# B&R Automation Studio project Y4_V3_1 (part 5)

#### ConBuffersCyclic.st - Cyclic code
```iecst
(********************************************************************
 * COPYRIGHT --
 ********************************************************************
 * Program: ConSeam2
 * File: ConSeam2Cyclic.st
 * Author: nicke
 ********************************************************************
 * Implementation of program ConSeam2
 ********************************************************************)

PROGRAM _CYCLIC

   //TRACKINGSECTION END BLOCK CONDITIONS
	Tracking30.Blocks[0] := (Tracking40.Busy) ;
	Tracking30.Blocks[2] := (CB2.Input.Fault) ;
	Tracking30.Blocks[9] := (S16Photo.Int) ;
	Tracking30.Blocks[10] := (S17Photo.Int) ;
	Tracking30.ControlIN := Control.Achieved1 ;
	Tracking30.EMOStart := EMO.StartLatch ;
	Tracking30.ESClear := Control.ESClear ;
	Tracking30 ();
	Tracking30.ResMan := FALSE ;
	Tracking30.BlockInhib := (Tracking41.Busy) AND NOT(Tracking40.Busy) ;
	CASE Tracking30.Index OF
		0: //RESET ALL TRACKBIT FOR SELECTED TRACKINGSECTION
			Track301 := TrackClear ;
			Track302 := TrackClear ;
		1: //TRACK FROM NOT Tracking20.Blocked (-) TO S14Photo.Int (P)
			Track302 := TrackClear ;
			//FB INPUTS
			Track301.FixedIN := Tracking30.FixedOUT ;
			Track301.Speed := Speeds.SpeedExit ;
			Track301.TimeoutEN := TRUE ;
			Track301.TimeoutACK := Warn.Ack ;
			Track301.TimeoutBlock := (Warn.Block) ;
			Track301.DelayPT := TrackDelayPT.PTTrack301 ;
			//FB CALL
			Track301 ();
			//FB OUTPUTS
			CB1.o.Run[0] := Track301.RunOUT ;
			CB1.Inv.Scale1.x := Track301.SpeedOUT ;
			IF(Track301.Done) THEN
				Tracking30.IndexIN := 2 ;
			END_IF
		2: //TRACK FROM S14Photo.Int (P) TO NOT Tracking30.Blocked (-)
			Track301 := TrackClear ;
			//FB INPUTS
			Track302.FixedIN := Tracking30.FixedOUT ;
			//FB CALL
			Track302 ();
			//FB OUTPUTS
			IF(Track302.Done) THEN
				Tracking30.IndexIN := 0 ;
				Tracking40.IndexIN := 1 ;
				Tracking93.IndexIN := 1 ;
				Tracking40.LengthIN := Tracking30.Length ;
				Tracking40.WidthIN := Tracking30.Width ;
				Tracking40.RowBlockIN := Tracking30.RowBlock ;
			END_IF
	END_CASE

	//TRACKBIT DONE CONDITIONS
	Track301.DoneIN := EDGEPOS(S14Photo.Int) ;
	Track302.DoneIN := NOT(Tracking30.Blocked) ;

	//TRACKINGSECTION END BLOCK CONDITIONS
	Tracking93.ControlIN := Control.Achieved1 ;
	Tracking93.EMOStart := EMO.StartLatch ;
	Tracking93.ESClear := Control.ESClear ;
	Tracking93 ();
	Tracking93.ResMan := FALSE ;
	CASE Tracking93.Index OF
		0: //RESET ALL TRACKBIT FOR SELECTED TRACKINGSECTION
			Track931 := TrackClear ;
			Track932 := TrackClear ;
		1: //TRACK FROM NOT Tracking30.Blocked (-) TO S15Photo.Int (N)
			Track932 := TrackClear ;
			//FB INPUTS
			Track931.FixedIN := Tracking93.FixedOUT ;
			Track931.RunBlock := (Track401.TimeoutOUT) OR(Track402.TimeoutOUT) ;
			Track931.Speed := Speeds.SpeedExit ;
			//FB CALL
			Track931 ();
			//FB OUTPUTS
			CB1.o.Run[0] := Track931.RunOUT ;
			CB1.Inv.Scale1.x := Track931.SpeedOUT ;
			IF(Track931.Done) THEN
				Tracking93.IndexIN := 2 ;
			END_IF
		2: //TRACK FROM S15Photo.Int (N) TO Track932.DelayTON.Q (P)
			Track931 := TrackClear ;
			//FB INPUTS
			Track932.FixedIN := Tracking93.FixedOUT ;
			Track932.RunBlock := (Track401.TimeoutOUT) OR(Track402.TimeoutOUT) ;
			Track932.Speed := Speeds.SpeedExit ;
			Track932.TrackDelayEN := TRUE ;
			Track932.DelayPT := TrackDelayPT.PTTrack932 ;
			//FB CALL
			Track932 ();
			//FB OUTPUTS
			CB1.o.Run[0] := Track932.RunOUT ;
			CB1.Inv.Scale1.x := Track932.SpeedOUT ;
			IF(Track932.Done) THEN
				Tracking93.IndexIN := 0 ;
			END_IF
	END_CASE

	//TRACKBIT DONE CONDITIONS
	Track931.DoneIN := EDGENEG(S15Photo.Int) ;

	//MANUAL RESET CONDITIONS FOR CONCURRENT TRACKBIT
	Tracking93.ResMan := Tracking40.ResMan ;
	IF(Tracking40.IndexIN = 0) THEN
		Tracking93.IndexIN := 0 ;
	END_IF
	IF EDGEPOS(Track302.Active)AND((Track401.Active)OR(Track402.Active))THEN
		Tracking93.IndexIN:=0;
	END_IF

	//TRACKINGSECTION END BLOCK CONDITIONS
	Tracking40.Blocks[0] := (Tracking41.Busy) OR(S58Lever.In ) OR(S58Lever.Int) OR(Tracking51.Busy) ;
	Tracking40.Blocks[1] := (Tracking50.IndexIN > 1) OR(Tracking52.Busy) ;
	Tracking40.Blocks[2] := (RowTemp.Done) ;
	Tracking40.Blocks[4] := NOT(Sol33Pal4.Auto) ;
	Tracking40.Blocks[9] := (S17Photo.Int) ;
	Tracking40.Blocks[10] := (S18Photo.Int) ;
	Tracking40.Blocks[11] := NOT(S37Reed.In) ;
	Tracking40.ControlIN := Control.Achieved1 ;
	Tracking40.EMOStart := EMO.StartLatch ;
	Tracking40.ESClear := Control.ESClear ;
	Tracking40 ();
	Tracking40.ResMan := FALSE ;
	CASE Tracking40.Index OF
		0: //RESET ALL TRACKBIT FOR SELECTED TRACKINGSECTION
			Track401 := TrackClear ;
			Track402 := TrackClear ;
		1: //TRACK FROM NOT Tracking30.Blocked (-) TO S16Photo.Int (P)
			Track402 := TrackClear ;
			//FB INPUTS
			Track401.FixedIN := Tracking40.FixedOUT ;
			Track401.Speed := Speeds.SpeedExit ;
			Track401.TimeoutEN := TRUE ;
			Track401.TimeoutACK := Warn.Ack ;
			Track401.TimeoutBlock := (Warn.Block) ;
			Track401.DelayPT := TrackDelayPT.PTTrack401 ;
			//FB CALL
			Track401 ();
			//FB OUTPUTS
			CB2.o.Run[0] := Track401.RunOUT ;
			CB2.Inv.Scale1.x := Track401.SpeedOUT ;
			IF(Track401.Done) THEN
				Tracking40.IndexIN := 2 ;
			END_IF
		2: //TRACK FROM S16Photo.Int (P) TO NOT Tracking40.Blocked (-)
			Track401 := TrackClear ;
			//FB INPUTS
			Track402.FixedIN := Tracking40.FixedOUT ;
			//FB CALL
			Track402 ();
			//FB OUTPUTS
			IF(Track402.Done) THEN
				Tracking40.IndexIN := 0 ;
				IF NOT(Tracking40.Blocked) THEN
					Tracking41.IndexIN := 1 ;
				ELSE
					Tracking41.IndexIN := 2 ;
				END_IF
				Tracking41.LengthIN := Tracking40.Length ;
				Tracking41.WidthIN := Tracking40.Width ;
				Tracking41.RowBlockIN := Tracking40.RowBlock ;
			END_IF
	END_CASE

	//TRACKBIT DONE CONDITIONS
	Track401.DoneIN := EDGEPOS(S16Photo.Int) ;
	Track402.DoneIN := NOT(Tracking40.Blocked) ;

	//TRACKINGSECTION END BLOCK CONDITIONS
	Tracking41.ControlIN := Control.Achieved1 ;
	Tracking41.EMOStart := EMO.StartLatch ;
	Tracking41.ESClear := Control.ESClear ;
	Tracking41 ();
	Tracking41.ResMan := FALSE ;
	CASE Tracking41.Index OF
		0: //RESET ALL TRACKBIT FOR SELECTED TRACKINGSECTION
			Track411 := TrackClear ;
			Track412 := TrackClear ;
			Track413 := TrackClear ;
			Track414 := TrackClear ;
		1: //TRACK FROM NOT Tracking40.Blocked (-) TO Track411.DelayTON.Q (P)
			Track412 := TrackClear ;
			Track413 := TrackClear ;
			Track414 := TrackClear ;
			//FB INPUTS
			Track411.FixedIN := Tracking41.FixedOUT ;
			Track411.Speed := Speeds.SpeedExit ;
			Track411.TrackDelayEN := TRUE ;
			Track411.DelayPT := TrackDelayPT.PTTrack411 ;
			//FB CALL
			Track411 ();
			//FB OUTPUTS
			CB2.o.Run[0] := Track411.RunOUT ;
			CB2.Inv.Scale1.x := Track411.SpeedOUT ;
			IF(Track411.Done) THEN
				Tracking41.IndexIN := 2 ;
			END_IF
		2: //TRACK FROM Track411.DelayTON.Q (P) TO S17Photo.Int (N)
			Track411 := TrackClear ;
			Track413 := TrackClear ;
			Track414 := TrackClear ;
			//FB INPUTS
			Track412.FixedIN := Tracking41.FixedOUT ;
			Track412.Speed := Speeds.SpeedExit ;
			Track412.TimeoutEN := TRUE ;
			Track412.TimeoutACK := Warn.Ack ;
			Track412.TimeoutBlock := (Warn.Block) ;
			Track412.DelayPT := TrackDelayPT.PTTrack412 ;
			//FB CALL
			Track412 ();
			//FB OUTPUTS
			CB2.o.Run[0] := Track412.RunOUT ;
			CRB.o.Run[0] := Track412.RunOUT ;
			CB2.Inv.Scale1.x := Track412.SpeedOUT ;
			CRB.Inv.Scale1.x := Track412.SpeedOUT ;
			IF(Track412.Done) THEN
				Tracking41.IndexIN := 3 ;
			END_IF
		3: //TRACK FROM S17Photo.Int (N) TO S17Photo.Int (P)
			Track411 := TrackClear ;
			Track412 := TrackClear ;
			Track414 := TrackClear ;
			//FB INPUTS
			Track413.FixedIN := Tracking41.FixedOUT ;
			Track413.Speed := Speeds.SpeedSlow ;
			Track413.TimeoutEN := TRUE ;
			Track413.TimeoutACK := Warn.Ack ;
			Track413.TimeoutBlock := (Warn.Block) ;
			Track413.DelayPT := TrackDelayPT.PTTrack413 ;
			//FB CALL
			Track413 ();
			//FB OUTPUTS
			CRB.o.Rev[0] := Track413.RunOUT ;
			CRB.Inv.Scale1.x := Track413.SpeedOUT ;
			IF(Track413.Done) THEN
				Tracking41.IndexIN := 4 ;
			END_IF
		4: //TRACK FROM S17Photo.Int (P) TO S17Photo.Int (N)
			Track411 := TrackClear ;
			Track412 := TrackClear ;
			Track413 := TrackClear ;
			//FB INPUTS
			Track414.FixedIN := Tracking41.FixedOUT ;
			Track414.Speed := Speeds.SpeedSlow ;
			//FB CALL
			Track414 ();
			//FB OUTPUTS
			CRB.o.Run[0] := Track414.RunOUT ;
			CRB.Inv.Scale1.x := Track414.SpeedOUT ;
			IF(Track414.Done) THEN
				Tracking41.IndexIN := 0 ;
				Tracking50.IndexIN := 1 ;
				Tracking50.RowBlockIN := Tracking41.RowBlock ;
			END_IF
	END_CASE

	//TRACKBIT DONE CONDITIONS
	Track412.DoneIN := EDGENEG(S17Photo.Int) ;
	Track413.DoneIN := EDGEPOS(S17Photo.Int) ;
	Track414.DoneIN := EDGENEG(S17Photo.Int) ;

END_PROGRAM
```

### Program Logical/Automatic/ConRow (IEC) - Row Building Conveyor

#### ConRowCyclic.st - Cyclic code
```iecst
(********************************************************************
 * COPYRIGHT --
 ********************************************************************
 * Program: ConRowBuild
 * File: ConRowBuildCyclic.st
 * Author: nicke
 ********************************************************************
 * Implementation of program ConRowBuild
 ********************************************************************)

PROGRAM _CYCLIC

   //TRACKINGSECTION END BLOCK CONDITIONS
	Tracking50.Blocks[0] := (Tracking60.Index > 1) ;
	Tracking50.Blocks[1] := Tracking70.Busy ;
	Tracking50.Blocks[2] := (CRE.Input.Fault) ;
	Tracking50.Blocks[3] := (CLB.Input.Fault) ;
	Tracking50.Blocks[9] := (S19Photo.Int) ;
//	Tracking50.Blocks[10] := (S20Photo.Int) ;
	Tracking50.Blocks[11] := (S21Photo.Int) ;
	Tracking50.ControlIN := Control.Achieved1 ;
	Tracking50.EMOStart := EMO.StartLatch ;
	Tracking50.ESClear := Control.ESClear ;
	Tracking50 ();
	IF(Tracking50.ResMan) OR(Tracking50.ResES) THEN
		Rows.Tracking50 := Rows.Empty ;
	END_IF
	Tracking50.ResMan := FALSE ;
	//RESET OF OUTPUTS
	Sol33Pal4.Auto := TRUE ;
	CASE Tracking50.Index OF
		0: //RESET ALL TRACKBIT FOR SELECTED TRACKINGSECTION
			Track501 := TrackClear ;
			Track502 := TrackClear ;
			Track503 := TrackClear ;
			Track504 := TrackClear ;
			Track505 := TrackClear ;
			Track506 := TrackClear ;
			Track507 := TrackClear ;
		1: //TRACK FROM S17Photo.Int (N) TO RowTemp.Done (P)
			Track502 := TrackClear ;
			Track503 := TrackClear ;
			Track504 := TrackClear ;
			Track505 := TrackClear ;
			Track506 := TrackClear ;
			Track507 := TrackClear ;
			//FB INPUTS
			Track501.FixedIN := Tracking50.FixedOUT ;
			//FB CALL
			Track501 ();
			//FB OUTPUTS
			IF(Track501.Done) THEN
				Tracking50.IndexIN := 2 ;
			END_IF
		2: //TRACK FROM RowTemp.Done (P) TO Track502.DelayTON.Q (P)
			Track501 := TrackClear ;
			Track503 := TrackClear ;
			Track504 := TrackClear ;
			Track505 := TrackClear ;
			Track506 := TrackClear ;
			Track507 := TrackClear ;
			//FB INPUTS
			Track502.FixedIN := Tracking50.FixedOUT ;
			Track502.Speed := Speeds.SpeedCntr ;
			Track502.TrackDelayEN := TRUE ;
			Track502.DelayPT := TrackDelayPT.PTTrack502 ;
			//FB CALL
			Track502 ();
			//FB OUTPUTS
			CRB.o.Run[0] := Track502.RunOUT ;
			CRB.Inv.Scale1.x := Track502.SpeedOUT ;
			IF(S18Photo.Int) THEN
				Track502.DoneIN := TRUE ;
			END_IF
			IF(Track502.Done) THEN
				IF NOT(Tracking50.RowBlock)THEN // Furnace 1
					Tracking50.IndexIN := 3 ;
				ELSE // Furnace 2
					Tracking50.IndexIN := 0 ;
					Tracking52.IndexIN := 3 ;
					Tracking52.LengthIN := Tracking50.Length ;
					Tracking52.BatchClearIN := Tracking50.BatchClear;
				END_IF
			END_IF
		3: //TRACK FROM Track502.DelayTON.Q (P) TO S36Reed.In (P)
			Track501 := TrackClear ;
			Track502 := TrackClear ;
			Track504 := TrackClear ;
			Track505 := TrackClear ;
			Track506 := TrackClear ;
			Track507 := TrackClear ;
			//FB INPUTS
			Track503.FixedIN := Tracking50.FixedOUT ;
			Track503.SolBlock := (Tracking50.Blocked) ;
			Track503.TimeoutEN := TRUE ;
			Track503.TimeoutACK := Warn.Ack ;
			Track503.TimeoutBlock := (Warn.Block) ;
			Track503.DelayPT := TrackDelayPT.PTTrack503 ;
			//FB CALL
			Track503 ();
			//FB OUTPUTS
			Sol33Pal4.Auto := NOT(Track503.SolOUT) ;
			IF(Track503.Done) THEN
				Tracking50.IndexIN := 4 ;
			END_IF
		4: //TRACK FROM S36Reed.In (P) TO S19Photo.Int (P)
			Track501 := TrackClear ;
			Track502 := TrackClear ;
			Track503 := TrackClear ;
			Track505 := TrackClear ;
			Track506 := TrackClear ;
			Track507 := TrackClear ;
			//FB INPUTS
			Track504.FixedIN := Tracking50.FixedOUT ;
			Track504.Speed := Speeds.SpeedBatch ;
			Track504.TimeoutEN := TRUE ;
			Track504.TimeoutACK := Warn.Ack ;
			Track504.TimeoutBlock := (Warn.Block) ;
			Track504.DelayPT := TrackDelayPT.PTTrack504 ;
			//FB CALL
			Track504 ();
			//FB OUTPUTS
			CRE.o.Run[0] := Track504.RunOUT ;
			CRE.Inv.Scale1.x := Track504.SpeedOUT ;
			Sol33Pal4.Auto := NOT(Track504.SolOUT) ;
			IF(Track504.Done) THEN
				Tracking50.IndexIN := 5 ;
			END_IF
		5: //TRACK FROM S19Photo.Int (P) TO Track505.DelayTON.Q (N)
			Track501 := TrackClear ;
			Track502 := TrackClear ;
			Track503 := TrackClear ;
			Track504 := TrackClear ;
			Track506 := TrackClear ;
			Track507 := TrackClear ;
			//FB INPUTS
			Track505.FixedIN := Tracking50.FixedOUT ;
			Track505.Speed := Speeds.SpeedBatch ;
			Track505.TrackDelayEN := TRUE ;
			Track505.DelayPT := TrackDelayPT.PTTrack505 ;
			//FB CALL
			Track505 ();
			//FB OUTPUTS
			CRE.o.Run[0] := Track505.RunOUT ;
			CRE.Inv.Scale1.x := Track505.SpeedOUT ;
			Sol33Pal4.Auto := NOT(Track505.SolOUT) ;
			IF(Track505.Done) THEN
				Tracking50.IndexIN := 6 ;
			END_IF
		6: //TRACK FROM Track505.DelayTON.Q (P) TO S19Photo.Int (N)
			Track501 := TrackClear ;
			Track502 := TrackClear ;
			Track503 := TrackClear ;
			Track504 := TrackClear ;
			Track505 := TrackClear ;
			Track507 := TrackClear ;
			//FB INPUTS
			Track506.FixedIN := Tracking50.FixedOUT ;
			Track506.Speed := Speeds.SpeedBatch ;
			Track506.TimeoutEN := TRUE ;
			Track506.TimeoutACK := Warn.Ack ;
			Track506.TimeoutBlock := (Warn.Block) ;
			Track506.DelayPT := TrackDelayPT.PTTrack506 ;
			//FB CALL
			Track506 ();
			//FB OUTPUTS
			CRE.o.Run[0] := Track506.RunOUT ;
			CLB.o.Run[0] := Track506.RunOUT ;
			CRE.Inv.Scale1.x := Track506.SpeedOUT ;
			CLB.Inv.Scale1.x := Track506.SpeedOUT ;
			Sol33Pal4.Auto := NOT(Track506.SolOUT) ;
			IF(Track506.Done) THEN
				Tracking50.IndexIN := 7 ;
			END_IF
		7: //TRACK FROM S19Photo.Int (N) TO Track507.DelayTON.Q (P)
			Track501 := TrackClear ;
			Track502 := TrackClear ;
			Track503 := TrackClear ;
			Track504 := TrackClear ;
			Track505 := TrackClear ;
			Track506 := TrackClear ;
			//FB INPUTS
			Track507.FixedIN := Tracking50.FixedOUT ;
			Track507.Speed := Speeds.SpeedSlow ;
			Track507.TrackDelayEN := TRUE ;
			Track507.DelayPT := TrackDelayPT.PTTrack507 ;
			//FB CALL
			Track507 ();
			//FB OUTPUTS
			CRE.o.Run[0] := Track507.RunOUT ;
			CLB.o.Run[0] := Track507.RunOUT ;
			CRE.Inv.Scale1.x := Track507.SpeedOUT ;
			CLB.Inv.Scale1.x := Track507.SpeedOUT ;
			IF(Track507.Done) THEN
				Tracking50.IndexIN := 0 ;
				Tracking60.IndexIN := 1 ;
				Tracking60.BatchClearIN := Tracking50.BatchClear ;
			END_IF
	END_CASE

	//TRACKBIT DONE CONDITIONS
	Track501.DoneIN := EDGEPOS(RowTemp.Done) ;
	Track503.DoneIN := EDGEPOS(S36Reed.In) ;
	Track504.DoneIN := EDGEPOS(S19Photo.Int) ;
	Track506.DoneIN := EDGENEG(S19Photo.Int) ;

	//TRACKINGSECTION END BLOCK CONDITIONS
	Tracking52.Blocks[0] := NOT(AGVReady.In) ;
	Tracking52.Blocks[1] := NOT(AGVInPosition.In) ;
	Tracking52.ControlIN := Control.Achieved1 ;
	Tracking52.EMOStart := EMO.StartLatch ;
	Tracking52.ESClear := Control.ESClear ;
	Tracking52 ();
	Tracking52.ResMan := FALSE ;
	//RESET OF OUTPUTS
	AGVReadyToSend.Auto := FALSE ;
	AGVSending.Auto := FALSE ;
	AGVBatchClear.Auto := FALSE;
	CASE Tracking52.Index OF
		0: //RESET ALL TRACKBIT FOR SELECTED TRACKINGSECTION
			Track521 := TrackClear ;
			Track522 := TrackClear ;
		1: //TRACK FROM Track502.DelayTON.Q (P) TO NOT(Tracking52.Blocked) (-)
			Track522 := TrackClear ;
			//FB INPUTS
			Track521.FixedIN := Tracking52.FixedOUT ;
			//FB CALL
			Track521 ();
			//FB OUTPUTS
			AGVReadyToSend.Auto := Track521.SolOUT ;
			IF(Track521.Done) THEN
				Tracking52.IndexIN := 2 ;
			END_IF
		2: //TRACK FROM NOT(Tracking52.Blocked) (-)  TO Track522.DelayTON.Q (P)
			Track521 := TrackClear ;
			//FB INPUTS
			Track522.FixedIN := Tracking52.FixedOUT ;
			//Track522.Speed := Speeds.SpeedBatch ; //SSS
			Track522.Speed := Speeds.SpeedTrans ; //SSS
			Track522.TrackDelayEN := TRUE ;
			Track522.DelayPT := TrackDelayPT.PTTrack805 ;
			//FB CALL
			Track522 ();
			//FB OUTPUTS
			AGVReadyToSend.Auto := Track522.SolOUT ;
			AGVSending.Auto := Track522.RunOUT ;
			AGVBatchClear.Auto := Tracking52.BatchClear;
			CRB.o.Run[0] := Track522.RunOUT ;
			CRB.Inv.Scale1.x := Track522.SpeedOUT ;
			IF(Track522.Done) THEN
				Tracking52.IndexIN := 0 ;
			END_IF
		3://Trick to beat the problem of Track521.DoneIN being true when IndexIN = 1.
			Tracking52.IndexIN := 1 ;
	END_CASE

	//TRACKBIT DONE CONDITIONS
	Track521.DoneIN := NOT(Tracking52.Blocked) ;

	AGVRequired.Auto := FALSE;
	IF(Tracking10.RowBlock) OR(Tracking11.RowBlock) OR(Tracking20.RowBlock) OR(Tracking30.RowBlock) OR(Tracking40.RowBlock) OR(Tracking50.RowBlock)THEN
		AGVRequired.Auto := TRUE;
	END_IF
END_PROGRAM
```

### Program Logical/Automatic/ConBatch (IEC) - Batch Building Conveyor

#### ConBatchCyclic.st - Cyclic code
```iecst
(********************************************************************
 * COPYRIGHT --
 ********************************************************************
 * Program: ConBatch
 * File: ConBatchCyclic.st
 * Author: nicke
 ********************************************************************
 * Implementation of program ConBatch
 ********************************************************************)

PROGRAM _CYCLIC

  //TRACKINGSECTION END BLOCK CONDITIONS
	Tracking60.Blocks[9] := (Pause.Active) ;
	Tracking60.Blocks[10] := NOT(WashRun.In) ;
	Tracking60.Blocks[11] := NOT(FurnReady.Int) ;
	Tracking60.Blocks[12] := (S55Lever.In) ;
	Tracking60.ControlIN := Control.Achieved1 ;
	Tracking60.EMOStart := EMO.StartLatch ;
	Tracking60.ESClear := Control.ESClear ;
	Tracking60 ();
	IF(Tracking60.ResMan) OR(Tracking60.ResES) THEN
		Loads.AshtonExit := Loads.Empty ;
	END_IF
	Tracking60.ResMan := FALSE ;
	//RESET OF OUTPUTS
	BatchAtExit.Auto := FALSE ;
	WashStop.Auto := FALSE ;
	CASE Tracking60.Index OF
		0: //RESET ALL TRACKBIT FOR SELECTED TRACKINGSECTION
			Track601 := TrackClear ;
			Track602 := TrackClear ;
			Track603 := TrackClear ;
		1: //TRACK FROM Track507.DelayTON.Q(Stop) (P) TO LoadTemp.Done (P)
			Track602 := TrackClear ;
			Track603 := TrackClear ;
			//FB INPUTS
			Track601.FixedIN := Tracking60.FixedOUT ;
			//FB CALL
			Track601 ();
			//FB OUTPUTS
			IF(Track601.Done) THEN
				Tracking60.IndexIN := 2 ;
			END_IF
		2: //TRACK FROM LoadTemp.Done (P) TO S21Photo.Int (P)
			Track601 := TrackClear ;
			Track603 := TrackClear ;
			//FB INPUTS
			Track602.FixedIN := Tracking60.FixedOUT ;
			Track602.Speed := Speeds.SpeedSlow ;
			Track602.TimeoutEN := TRUE ;
			Track602.TimeoutACK := Warn.Ack ;
			Track602.TimeoutBlock := (Warn.Block) ;
			Track602.DelayPT := TrackDelayPT.PTTrack602 ;
			//FB CALL
			Track602 ();
			//FB OUTPUTS
			CLB.o.Run[0] := Track602.RunOUT ;
			CLB.Inv.Scale1.x := Track602.SpeedOUT ;
			IF(Track602.Done) THEN
				Tracking60.IndexIN := 3 ;
			END_IF
		3: //TRACK FROM S21Photo.Int (P) TO NOT(Tracking60.Blocked) (-)
			Track601 := TrackClear ;
			Track602 := TrackClear ;
			//FB INPUTS
			Track603.FixedIN := Tracking60.FixedOUT ;
			Track603.SolBlock := (S55Lever.In)OR NOT(WashRun.In) ;
			//FB CALL
			Track603 ();
			//FB OUTPUTS
			BatchAtExit.Auto := (Track603.SolOUT) ;
			IF(Track603.Done) THEN
				Tracking60.IndexIN := 0 ;
				Tracking70.IndexIN := 1 ;
			END_IF
	END_CASE

	//TRACKBIT DONE CONDITIONS
	Track601.DoneIN := EDGEPOS(LoadTemp.Done) ;
	Track602.DoneIN := (S21Photo.Int) ;
	Track603.DoneIN := NOT(Tracking60.Blocked) ;

	//TRACKINGSECTION END BLOCK CONDITIONS
	Tracking70.ControlIN := Control.Achieved1 ;
	Tracking70.EMOStart := EMO.StartLatch ;
	Tracking70.ESClear := Control.ESClear ;
	Tracking70 ();
	Tracking70.ResMan := FALSE ;
	IF(CLB.LastSpeed = 0.0)THEN
		TrackDelayPT.PTTrack601 := 1000 ;
	ELSE
		TrackDelayPT.PTTrack601	:=	REAL_TO_UDINT((UDINT_TO_REAL(TrackDelayPT.PTTrack701)) *((10/CLB.LastSpeed)));
	END_IF
	CASE Tracking70.Index OF
		0: //RESET ALL TRACKBIT FOR SELECTED TRACKINGSECTION
			Track701 := TrackClear ;
		1: //TRACK FROM NOT(Tracking60.Blocked) (-) TO Track701.DelayTON.Q (P)
			//FB INPUTS
			Track701.FixedIN := Tracking70.FixedOUT ;
			Track701.Speed := Speeds.SpeedWash ;
			Track701.Analog := InvPerms.CLB.Analog ;
			Track701.SpeedAnalog := CLB.SpeedAnalog ;
			Track701.TrackDelayEN := TRUE ;
			Track701.DelayPT := TrackDelayPT.PTTrack601 ;
			//FB CALL
			Track701 ();
			//FB OUTPUTS
			CLB.o.Run[0] := Track701.RunOUT ;
			CLB.Inv.Scale1.x := Track701.SpeedOUT ;
			BatchAtExit.Auto := (Track701.SolOUT) ;
			WashStop.Auto := Track701.RunOUT ;
			IF(Track701.Done) THEN
				Tracking70.IndexIN := 0 ;
			END_IF
	END_CASE

END_PROGRAM
```

### Program Logical/Automatic/Seaming (IEC)

#### Main.st - Cyclic code
```iecst
PROGRAM _CYCLIC

	//SEAMER 1
	IF (ProcessMode.In) THEN
		//BELT 1 TIMING CONTROL
		Belt1.PT_On := TrackDelayPT.PTTrack004 ;
		Belt1.PT_Off := TrackDelayPT.PTTrack103 ;
		//BELT 2 TIMING CONTROL
		Belt2.PT_On := TrackDelayPT.PTTrack005 ;
		Belt2.PT_Off :=  TrackDelayPT.PTTrack108 ;
		//BELT 3 TIMING CONTROL
		Belt3.PT_On := TrackDelayPT.PTTrack012 ;
		Belt3.PT_Off := TrackDelayPT.PTTrack114 ;
		//BELT 4 TIMING CONTROL
		Belt4.PT_On := TrackDelayPT.PTTrack013 ;
		Belt4.PT_Off :=  TrackDelayPT.PTTrack115 ;
	ELSE
		//BELT 1 TIMING CONTROL
		Belt1.PT_On := PresetSeam.BeltOn[1] ;
		Belt1.PT_Off := PresetSeam.BeltOff[1] ;
		//BELT 2 TIMING CONTROL
		Belt2.PT_On := PresetSeam.BeltOn[2] ;
		Belt2.PT_Off :=  PresetSeam.BeltOff[2] ;
		//BELT 3 TIMING CONTROL
		Belt3.PT_On := PresetSeam.BeltOn[3] ;
		Belt3.PT_Off := PresetSeam.BeltOff[3] ;
		//BELT 4 TIMING CONTROL
		Belt4.PT_On := PresetSeam.BeltOn[4] ;
		Belt4.PT_Off :=  PresetSeam.BeltOff[4] ;
	END_IF
	Belt1 ();
	Belt2 ();
	Belt3 ();
	Belt4 ();

	//START DELAY BEFORE ON
	IF EDGEPOS(Seaming.Start1) AND(Control.Achieved1) THEN
		Belt1.ONStart := TRUE ;
		Belt2.ONStart := TRUE ;
		Belt3.ONStart := TRUE ;
		Belt4.ONStart := TRUE ;
	ELSE
		Belt1.ONStart := FALSE ;
		Belt2.ONStart := FALSE ;
		Belt3.ONStart := FALSE ;
		Belt4.ONStart := FALSE ;
	END_IF
	//START DELAY BEFORE OFF
	IF EDGEPOS(Seaming.Stop1) AND(Control.Achieved1) THEN
		Belt1.OFFStart := TRUE ;
		Belt2.OFFStart := TRUE ;
		Belt3.OFFStart := TRUE ;
		Belt4.OFFStart := TRUE ;
	ELSE
		Belt1.OFFStart :=  FALSE ;
		Belt2.OFFStart := FALSE ;
		Belt3.OFFStart :=  FALSE ;
		Belt4.OFFStart := FALSE ;
	END_IF
	//ESTOP INPUT
	IF(Control.ESClear) OR(EMO.StartLatch) THEN
		Belt1.EStop := TRUE ;
		Belt2.EStop := TRUE ;
		Belt3.EStop := TRUE ;
		Belt4.EStop := TRUE ;
	ELSE
		Belt1.EStop := FALSE ;
		Belt2.EStop := FALSE ;
		Belt3.EStop := FALSE ;
		Belt4.EStop := FALSE ;
	END_IF
	//END CONDITIONS
	IF EDGENEG(Track104.Done) THEN
		Belt1.End := TRUE ;
		Belt2.End := TRUE ;
		Belt3.End := TRUE ;
		Belt4.End := TRUE ;
	ELSE
		Belt1.End := FALSE ;
		Belt2.End := FALSE ;
		Belt3.End := FALSE ;
		Belt4.End := FALSE ;
	END_IF
	//OUTPUTS
	IF(SeamersII.Enable[1]) THEN
		IF(Belt1.Out) AND NOT(Control.ESClear) THEN
			Sol1Blt1.Auto := TRUE ;
		ELSE
			Sol1Blt1.Auto := FALSE ;
		END_IF
		IF(Belt2.Out) AND NOT(Control.ESClear) THEN
			Sol2Blt2.Auto := TRUE ;
		ELSE
			Sol2Blt2.Auto := FALSE ;
		END_IF
		IF(Belt3.Out) AND NOT(Control.ESClear) THEN
			Sol3Blt3.Auto := TRUE ;
		ELSE
			Sol3Blt3.Auto := FALSE ;
		END_IF
		IF(Belt4.Out) AND NOT(Control.ESClear) THEN
			Sol4Blt4.Auto := TRUE ;
		ELSE
			Sol4Blt4.Auto := FALSE ;
		END_IF
	END_IF
	//CALCULATION OF BELTS COMPLETE
	IF NOT(Seaming.Stop1) THEN
		Belts1.Done := FALSE ;
		Belts1.Start := FALSE ;
	END_IF
	IF(Seaming.Stop1) AND(Control.Achieved1) THEN
		Belts1.Start := TRUE ;
	END_IF
	IF (Belts1.Start)THEN
		IF NOT((Belt1.Out) OR(Belt2.Out) OR(Belt3.Out) OR(Belt4.Out)) THEN
			Belts1.Done := TRUE ;
		END_IF
	END_IF

	//SEAMER 2
	IF (ProcessMode.In) THEN
		//BELT 5 TIMING CONTROL
		Belt5.PT_On := TrackDelayPT.PTTrack203 ;
		Belt5.PT_Off := TrackDelayPT.PTTrack501 ;
		//BELT 6 TIMING CONTROL
		Belt6.PT_On := TrackDelayPT.PTTrack208 ;
		Belt6.PT_Off :=  TrackDelayPT.PTTrack901 ;
		//BELT 7 TIMING CONTROL
		Belt7.PT_On := TrackDelayPT.PTTrack302 ;
		Belt7.PT_Off := TrackDelayPT.PTTrack911 ;
		//BELT 8 TIMING CONTROL
		Belt8.PT_On := TrackDelayPT.PTTrack402 ;
		Belt8.PT_Off :=  TrackDelayPT.PTTrack912 ;
	ELSE
		//BELT 5 TIMING CONTROL
		Belt5.PT_On := PresetSeam.BeltOn[5] ;
		Belt5.PT_Off := PresetSeam.BeltOff[5] ;
		//BELT 6 TIMING CONTROL
		Belt6.PT_On := PresetSeam.BeltOn[6] ;
		Belt6.PT_Off :=  PresetSeam.BeltOff[6] ;
		//BELT 7 TIMING CONTROL
		Belt7.PT_On := PresetSeam.BeltOn[7] ;
		Belt7.PT_Off := PresetSeam.BeltOff[7] ;
		//BELT 8 TIMING CONTROL
		Belt8.PT_On := PresetSeam.BeltOn[8] ;
		Belt8.PT_Off :=  PresetSeam.BeltOff[8] ;
	END_IF
	Belt5 ();
	Belt6 ();
	Belt7 ();
	Belt8 ();

	//START DELAY BEFORE ON
	IF EDGEPOS(Seaming.Start2) AND(Control.Achieved1) THEN
		Belt5.ONStart := TRUE ;
		Belt6.ONStart := TRUE ;
		Belt7.ONStart := TRUE ;
		Belt8.ONStart := TRUE ;
	ELSE
		Belt5.ONStart := FALSE ;
		Belt6.ONStart := FALSE ;
		Belt7.ONStart := FALSE ;
		Belt8.ONStart := FALSE ;
	END_IF
	//START DELAY BEFORE OFF
	IF EDGEPOS(Seaming.Stop2) AND(Control.Achieved1) THEN
		Belt5.OFFStart := TRUE ;
		Belt6.OFFStart := TRUE ;
		Belt7.OFFStart := TRUE ;
		Belt8.OFFStart := TRUE ;
	ELSE
		Belt5.OFFStart :=  FALSE ;
		Belt6.OFFStart := FALSE ;
		Belt7.OFFStart :=  FALSE ;
		Belt8.OFFStart := FALSE ;
	END_IF
	//ESTOP INPUT
	IF(Control.ESClear) OR(EMO.StartLatch) THEN
		Belt5.EStop := TRUE ;
		Belt6.EStop := TRUE ;
		Belt7.EStop := TRUE ;
		Belt8.EStop := TRUE ;
	ELSE
		Belt5.EStop := FALSE ;
		Belt6.EStop := FALSE ;
		Belt7.EStop := FALSE ;
		Belt8.EStop := FALSE ;
	END_IF
	//END CONDITIONS
	IF EDGENEG(Track204.Done) THEN
		Belt5.End := TRUE ;
		Belt6.End := TRUE ;
		Belt7.End := TRUE ;
		Belt8.End := TRUE ;
	ELSE
		Belt5.End := FALSE ;
		Belt6.End := FALSE ;
		Belt7.End := FALSE ;
		Belt8.End := FALSE ;
	END_IF
	//OUTPUTS
	IF(SeamersII.Enable[2]) THEN
		IF(Belt5.Out) AND NOT(Control.ESClear) THEN
			Sol10Blt5.Auto := TRUE ;
		ELSE
			Sol10Blt5.Auto := FALSE ;
		END_IF
		IF(Belt6.Out) AND NOT(Control.ESClear) THEN
			Sol11Blt6.Auto := TRUE ;
		ELSE
			Sol11Blt6.Auto := FALSE ;
		END_IF
		IF(Belt7.Out) AND NOT(Control.ESClear) THEN
			Sol12Blt7.Auto := TRUE ;
		ELSE
			Sol12Blt7.Auto := FALSE ;
		END_IF
		IF(Belt8.Out) AND NOT(Control.ESClear) THEN
			Sol13Blt8.Auto := TRUE ;
		ELSE
			Sol13Blt8.Auto := FALSE ;
		END_IF
	END_IF
	//CALCULATION OF BELTS COMPLETE
	IF NOT(Seaming.Stop2) THEN
		Belts2.Done := FALSE ;
		Belts2.Start := FALSE ;
	END_IF
	IF(Seaming.Stop2) AND(Control.Achieved1) THEN
		Belts2.Start := TRUE ;
	END_IF
	IF (Belts2.Start)THEN
		IF NOT((Belt5.Out) OR(Belt6.Out) OR(Belt7.Out) OR(Belt8.Out)) THEN
			Belts2.Done := TRUE ;
		END_IF
	END_IF

	//SECTION TO INHIBIT INDIVIDUAL EDGE GRINDING
	IF(SeamBlock[1]) THEN
		Sol1Blt1.Auto := FALSE ;
		Sol2Blt2.Auto := FALSE ;
	END_IF
	IF(SeamBlock[2]) THEN
		Sol3Blt3.Auto := FALSE ;
		Sol4Blt4.Auto := FALSE ;
	END_IF
	IF(SeamBlock[3]) THEN
		Sol10Blt5.Auto := FALSE ;
		Sol11Blt6.Auto := FALSE ;
	END_IF
	IF(SeamBlock[4]) THEN
		Sol12Blt7.Auto := FALSE ;
		Sol13Blt8.Auto := FALSE ;
	END_IF

END_PROGRAM
```

### Program Logical/Automatic/Batching (IEC)

#### Cyclic.st
```iecst
PROGRAM _CYCLIC

	//ROW COMPLETION AND CENTERING CALCULATIONS
	//FB INPUTS
	RowTemp.Type := ROW ;
	RowTemp.Calculate := (Track414.Active) AND NOT(Control.ESClear) ;
	RowTemp.Building := (Track501.Active) OR(Track502.Active) ;
	RowTemp.FollowingIN[0] := Tracking41.Width ;
	RowTemp.FollowingIN[1] := Tracking40.Width ;
	RowTemp.FollowingIN[2] := Tracking30.Width ;
	RowTemp.FollowingIN[3] := Tracking20.Width ;
	RowTemp.LengthIN := Tracking41.Length ;
	RowTemp.Gap := RowPerm.Gap ;
	RowTemp.MaxSize := RowPerm.Max ;
	RowTemp.CenterDist := RowPerm.CenterDist ;
	RowTemp.CenterSpeed := Speeds.SpeedCntr ;
	RowTemp.ClearIN := (ClearBatch.In) OR(RowTemp.ClearIN);
	IF(RowTemp.ClearIN) AND(Track501.Active)THEN
		Tracking50.BatchClearIN := TRUE	;
	ELSIF(RowTemp.ClearIN) AND(Track601.Active) AND NOT(Tracking50.Busy) THEN
		Tracking60.BatchClearIN := TRUE ;
		RowTemp.ClearIN := FALSE ;
	END_IF
	// Clear Row if Furnace 2 switched to Furnace 1
	IF(Track501.Active) AND(Tracking50.RowBlock)THEN
		IF(Tracking20.Width > 0.0) AND NOT(Tracking20.RowBlock)THEN
			RowTemp.ClearIN := TRUE	;
			Tracking50.BatchClearIN := TRUE	;
		ELSIF(Tracking30.Width > 0.0) AND NOT(Tracking30.RowBlock)THEN
			RowTemp.ClearIN := TRUE	;
			Tracking50.BatchClearIN := TRUE	;
		ELSIF(Tracking40.Width > 0.0) AND NOT(Tracking40.RowBlock)THEN
			RowTemp.ClearIN := TRUE	;
			Tracking50.BatchClearIN := TRUE	;
		END_IF
	END_IF
	// Clear row if Furnace 1 switched to Furnace 2
	IF(Track501.Active) AND NOT(Tracking50.RowBlock)THEN
		IF(Tracking20.Width > 0.0) AND(Tracking20.RowBlock)THEN
			RowTemp.ClearIN := TRUE	;
			Tracking50.BatchClearIN := TRUE	;
		ELSIF(Tracking30.Width > 0.0) AND(Tracking30.RowBlock)THEN
			RowTemp.ClearIN := TRUE	;
			Tracking50.BatchClearIN := TRUE	;
		ELSIF(Tracking40.Width > 0.0) AND(Tracking40.RowBlock)THEN
			RowTemp.ClearIN := TRUE	;
			Tracking50.BatchClearIN := TRUE	;
		END_IF
	END_IF
	//CALL FB
	RowTemp ();
	RowTemp.ClearIN := FALSE ;
	//FB OUTPUTS
	TrackDelayPT.PTTrack502 := RowTemp.CenterPT ;
	IF(RowTemp.Building) THEN
		Tracking50.WidthIN := RowTemp.Current ;
		Tracking50.LengthIN := RowTemp.Longest ;
	END_IF

	//LOAD COMPLETION CALCULATIONS
	//FB INPUTS
	LoadTemp.Type := LOAD ;
	LoadTemp.Calculate := (Track507.Active) AND NOT(Control.ESClear) ;
	LoadTemp.Building := (Track601.Active) OR(Track602.Active) ;
	LoadTemp.FollowingIN[0] := Tracking50.Length ;
	LoadTemp.Gap := LoadPerm.Gap ;
	LoadTemp.MaxSize := LoadPerm.Max ;
	LoadTemp.ClearIN := Tracking60.BatchClear ;
	//CALL FB
	LoadTemp ();
	//FB OUTPUTS
	IF EDGENEG(LoadTemp.Building) THEN
		LoadTemp.ClearIN := FALSE ;
	END_IF

	//BATCH DISPLAY DATA
	IF EDGEPOS(Track414.Done) AND NOT(Tracking41.RowBlock) THEN
		Rows.Tracking50.Row[DataFlow.IndexRow].Width:=Tracking41.Width;
		Rows.Tracking50.Row[DataFlow.IndexRow].Length:=Tracking41.Length;
		Rows.Tracking50.NotEmpty:=TRUE;
		DataFlow.IndexRow:=DataFlow.IndexRow+1;
	END_IF

	IF EDGEPOS(Track503.Done)THEN
		DataFlow.IndexRow:=1;
	END_IF

	IF EDGEPOS(Track507.Done) THEN
		Rows.Tracking50.Row[0].Width:= Tracking50.Width;
		Rows.Tracking50.Row[0].Length:= Tracking50.Length;
		Loads.AshtonExit.Rows[DataFlow.IndexLoad]:=Rows.Tracking50;
		Loads.AshtonExit.NotEmpty:=TRUE;
		DataFlow.IndexLoad:=DataFlow.IndexLoad+1;
		Rows.Tracking50:=Rows.Empty;
	END_IF

	IF EDGEPOS(Track603.Done)THEN
		IF NOT(Loads.Furnace9.NotEmpty)THEN
			Loads.Furnace9:=Loads.AshtonExit;
			Loads.AshtonExit:=Loads.Empty;
		ELSIF NOT(Loads.Furnace8.NotEmpty)THEN
			Loads.Furnace8:=Loads.AshtonExit;
			Loads.AshtonExit:=Loads.Empty;
		ELSIF NOT(Loads.Furnace7.NotEmpty)THEN
			Loads.Furnace7:=Loads.AshtonExit;
			Loads.AshtonExit:=Loads.Empty;
		ELSIF NOT(Loads.Furnace6.NotEmpty)THEN
			Loads.Furnace6:=Loads.AshtonExit;
			Loads.AshtonExit:=Loads.Empty;
		ELSIF NOT(Loads.Furnace5.NotEmpty)THEN
			Loads.Furnace5:=Loads.AshtonExit;
			Loads.AshtonExit:=Loads.Empty;
		ELSIF NOT(Loads.Furnace4.NotEmpty)THEN
			Loads.Furnace4:=Loads.AshtonExit;
			Loads.AshtonExit:=Loads.Empty;
		ELSIF NOT(Loads.Furnace3.NotEmpty)THEN
			Loads.Furnace3:=Loads.AshtonExit;
			Loads.AshtonExit:=Loads.Empty;
		ELSIF NOT(Loads.Furnace2.NotEmpty)THEN
			Loads.Furnace2:=Loads.AshtonExit;
			Loads.AshtonExit:=Loads.Empty;
		ELSIF NOT(Loads.Furnace1.NotEmpty)THEN
			Loads.Furnace1:=Loads.AshtonExit;
			Loads.AshtonExit:=Loads.Empty;
		END_IF
		DataFlow.IndexLoad:=1;
	END_IF

	//Encode size information to send to AGV controller
	IF EDGEPOS(Track414.Done) AND(Tracking41.RowBlock) THEN
		SizeData.CurrentWidth := REAL_TO_UINT(Tracking41.Width);
		SizeData.CurrentLength := REAL_TO_UINT(Tracking41.Length);
	END_IF

	CASE SizeData.Sequence OF
		SD_Idle:
			SizeData.WidthMask := FALSE;
			SizeData.LengthMask := FALSE;
			IF(SizeData.CurrentWidth > 0)THEN
				SizeData.Sequence := SD_WidthData;
			END_IF
		SD_WidthData:
			FOR i := 0 TO 11 DO
				SizeData.Sizes[i] := (SHR(SizeData.CurrentWidth, i) AND 1) <> 0;
			END_FOR
			SizeData.WidthMask := TRUE;
			SizeData.Sequence := SD_WidthACK;
		SD_WidthACK:
			IF(AGVAcknowledge.In)THEN
				SizeData.Sequence := SD_NotWidthACK;
				SizeData.WidthMask := FALSE;
				SizeData.CurrentWidth := 0;
			END_IF
		SD_NotWidthACK:
			IF NOT(AGVAcknowledge.In)THEN
				SizeData.Sequence := SD_LengthData;
			END_IF
		SD_LengthData:
			FOR i := 0 TO 11 DO
				SizeData.Sizes[i] := (SHR(SizeData.CurrentLength, i) AND 1) <> 0;
			END_FOR
			SizeData.LengthMask := TRUE;
			SizeData.Sequence := SD_LengthACK;
		SD_LengthACK:
			IF(AGVAcknowledge.In)THEN
				SizeData.Sequence := SD_NotLengthACK;
				SizeData.LengthMask := FALSE;
				SizeData.CurrentLength := 0;
			END_IF
		SD_NotLengthACK:
			IF NOT(AGVAcknowledge.In)THEN
				SizeData.Sequence := SD_Idle;
			END_IF
	END_CASE

END_PROGRAM
```

### Program Logical/Automatic/Modes (IEC) - Mode options program

#### ModesCyclic.st - Cyclic code
```iecst
(********************************************************************
 * COPYRIGHT --
 ********************************************************************
 * Program: Modes
 * File: ModesCyclic.st
 * Author: NE
 ********************************************************************)

PROGRAM _CYCLIC

	//LINE PAUSE - AT EXIT
	//BLOCK EXIT FROM CLB IF FURNACE LOAD CONVEYOR NOT CLEAR
	IF EDGEPOS(Perms.FurnReady = 0) THEN
		FurnReady.Int := FALSE ;
	END_IF
	Perms.FurnReady := 1 ;
	CASE Perms.FurnReady OF
		0:	//PULSE SIGNAL FROM FURNACE
			//CAPTURE FURNACE CLEAR SIGNAL
			IF EDGEPOS(FurnReady.In) THEN
				FurnReady.Int := TRUE ;
			END_IF
			IF EDGENEG(Track701.Active) AND NOT(Control.ESClear) THEN
				FurnReady.Int := FALSE ;
			END_IF
			IF EDGENEG(Track822.Active) AND NOT(Control.ESClear) THEN
				FurnReady.Int := FALSE ;
			END_IF
		1:	//ON SIGNAL FROM FURNACE
			Pause.Clear1.PT := t#500ms;//USE Pause Mode_typ spare variables to filter furnace input signal.
			Pause.Clear1.IN := FurnReady.In;
			Pause.Clear1 ();
			FurnReady.Int := Pause.Clear1.Q;
			IF EDGEPOS(FurnReady.In)THEN
				Pause.ESDisp := Pause.ESDisp + 1;
			END_IF
			IF EDGEPOS(Pause.Clear1.Q)THEN
				Pause.ESDisp := Pause.ESDisp - 1;
			END_IF
			Pause.ESDisp := LIMIT(0, Pause.ESDisp, 250);
	END_CASE

	//PAUSE CONDITIONS
	Pause.Input1 := S55Lever.In ;
	Pause.Input2 := NOT(WashRun.In) ;
	Pause.Input3 := NOT(FurnReady.Int) ;
	Pause.Input4 := FALSE ;

	IF(Track603.Active) OR(Track812.Active) OR(Track513.Active) THEN
		IF(Pause.Input1) OR(Pause.Input2) OR(Pause.Input3) OR(Pause.Input4) THEN
			Pause.Active	:=	TRUE	;
		END_IF
	END_IF

	//LINE PAUSE RESET
	IF EDGENEG(Pause.Input1) AND NOT(Pause.Input2) AND NOT(Pause.Input3) AND NOT(Pause.Input4) AND(Pause.Active) THEN
		Pause.Active	:= 	FALSE	;
	END_IF

	IF EDGENEG(Pause.Input2) AND NOT(Pause.Input1) AND NOT(Pause.Input3) AND NOT(Pause.Input4) AND(Pause.Active) THEN
		Pause.Active	:= 	FALSE	;
	END_IF

	IF EDGENEG(Pause.Input3) AND NOT(Pause.Input1) AND NOT(Pause.Input2) AND NOT(Pause.Input4) AND(Pause.Active) THEN
		Pause.Active	:= 	FALSE	;
	END_IF

	IF EDGENEG(Pause.Input4) AND NOT(Pause.Input1) AND NOT(Pause.Input2) AND NOT(Pause.Input3) AND(Pause.Active) THEN
		Pause.Active	:= 	FALSE	;
	END_IF

	IF NOT(Track603.Active) AND NOT(Track812.Active) AND NOT(Track513.Active) THEN
		Pause.Active	:=	FALSE	;
	END_IF

	//TRACKINGSECTION END BLOCK CONDITIONS
	Tracking80.Blocks[1] := (Tracking82.Busy) ;
	Tracking80.Blocks[2] := (CLB.Input.Fault) ;
	Tracking80.Blocks[9] := (S19Photo.Int) ;
	Tracking80.ControlIN := Control.Achieved1 ;
	Tracking80.EMOStart := EMO.StartLatch ;
	Tracking80.ESClear := Control.ESClear ;
	Tracking80 ();
	Tracking80.ResMan := FALSE ;
	IF(S57Lever.In) AND NOT((Tracking41.Busy) OR(Tracking50.Busy) OR(Tracking60.Busy) OR(Tracking70.Busy)) THEN
		S57Lever.Int := TRUE ;
	END_IF
	IF NOT(S57Lever.In) AND NOT((Tracking70.Busy) OR(Tracking80.Busy) OR(Tracking81.Busy) OR(Tracking82.Busy)) THEN
		S57Lever.Int := FALSE ;
	END_IF
	CASE Tracking80.Index OF
		0: //RESET ALL TRACKBIT FOR SELECTED TRACKINGSECTION
			Track801 := TrackClear ;
			Track802 := TrackClear ;
			Track803 := TrackClear ;
			Track804 := TrackClear ;
			Track805 := TrackClear ;
			//START CONDITION FOR LOADING
			IF((S18Photo.Int) AND(S57Lever.Int) AND(S37Reed.In) AND NOT(Tracking81.Busy) AND(Control.Achieved1)) THEN
				Tracking80.IndexIN := 1 ;
			END_IF
		1: //TRACK FROM S18Photo.Int (P) TO S18Photo.Int (N)
			Track802 := TrackClear ;
			Track803 := TrackClear ;
			Track804 := TrackClear ;
			Track805 := TrackClear ;
			//FB INPUTS
			Track801.FixedIN := Tracking80.FixedOUT ;
			Track801.Speed := Speeds.SpeedEntry ;
			Track801.TimeoutEN := TRUE ;
			Track801.TimeoutACK := Warn.Ack ;
			Track801.TimeoutBlock := (Warn.Block) ;
			Track801.DelayPT := TrackDelayPT.PTTrack801 ;
			//FB CALL
			Track801 ();
			//FB OUTPUTS
			CRB.o.Rev[0] := Track801.RunOUT ;
			CRB.Inv.Scale1.x := Track801.SpeedOUT ;
			IF(Track801.Done) THEN
				Tracking80.IndexIN := 2 ;
			END_IF
		2: //TRACK FROM S18Photo.Int (N) TO Track802.DelayTON.Q (P)
			Track801 := TrackClear ;
			Track803 := TrackClear ;
			Track804 := TrackClear ;
			Track805 := TrackClear ;
			//FB INPUTS
			Track802.FixedIN := Tracking80.FixedOUT ;
			Track802.Speed := Speeds.SpeedEntry ;
			Track802.TrackDelayEN := TRUE ;
			Track802.DelayPT := TrackDelayPT.PTTrack802 ;
			//FB CALL
			Track802 ();
			//FB OUTPUTS
			CRB.o.Rev[0] := Track802.RunOUT ;
			CRB.Inv.Scale1.x := Track802.SpeedOUT ;
			IF(Track802.Done) THEN
				Tracking80.IndexIN := 3 ;
			END_IF
		3: //TRACK FROM Track802.DelayTON.Q (P) TO S36Reed.In (P)
			Track801 := TrackClear ;
			Track802 := TrackClear ;
			Track804 := TrackClear ;
			Track805 := TrackClear ;
			//FB INPUTS
			Track803.FixedIN := Tracking80.FixedOUT ;
			Track803.SolBlock := (Tracking80.Blocked) ;
			Track803.TimeoutEN := TRUE ;
			Track803.TimeoutACK := Warn.Ack ;
			Track803.TimeoutBlock := (Warn.Block) ;
			Track803.DelayPT := TrackDelayPT.PTTrack803 ;
			//FB CALL
			Track803 ();
			//FB OUTPUTS
			Sol33Pal4.Auto := NOT(Track803.SolOUT) ;
			IF(Track803.Done) THEN
				Tracking80.IndexIN := 4 ;
			END_IF
		4: //TRACK FROM S36Reed.In (P) TO S19Photo.Int (P)
			Track801 := TrackClear ;
			Track802 := TrackClear ;
			Track803 := TrackClear ;
			Track805 := TrackClear ;
			//FB INPUTS
			Track804.FixedIN := Tracking80.FixedOUT ;
			Track804.Speed := Speeds.SpeedBatch ;
			Track804.TimeoutEN := TRUE ;
			Track804.DelayPT := TrackDelayPT.PTTrack804 ;
			//FB CALL
			Track804 ();
			//FB OUTPUTS
			CRE.o.Run[0] := Track804.RunOUT ;
			CLB.o.Run[0] := Track804.RunOUT ;
			CRE.Inv.Scale1.x := Track804.SpeedOUT ;
			CLB.Inv.Scale1.x := Track804.SpeedOUT ;
			Sol33Pal4.Auto := NOT(Track804.SolOUT) ;
			IF(Track804.TimeoutOUT) THEN
				Tracking80.IndexIN := 0 ;
			END_IF
			IF(Track804.Done) THEN
				Tracking80.IndexIN := 5 ;
			END_IF
		5: //TRACK FROM S19Photo.Int (P) TO S19Photo.Int (N)
			Track801 := TrackClear ;
			Track802 := TrackClear ;
			Track803 := TrackClear ;
			Track804 := TrackClear ;
			//FB INPUTS
			Track805.FixedIN := Tracking80.FixedOUT ;
			Track805.Speed := Speeds.SpeedBatch ;
			//FB CALL
			Track805 ();
			//FB OUTPUTS
			CRE.o.Run[0] := Track805.RunOUT ;
			CLB.o.Run[0] := Track805.RunOUT ;
			CRE.Inv.Scale1.x := Track805.SpeedOUT ;
			CLB.Inv.Scale1.x := Track805.SpeedOUT ;
			Sol33Pal4.Auto := NOT(Track805.SolOUT) ;
			IF(Track805.Done) THEN
				Tracking80.IndexIN := 0 ;
				Tracking81.IndexIN := 1 ;
			END_IF
	END_CASE

	//TRACKBIT DONE CONDITIONS
	Track801.DoneIN := EDGENEG(S18Photo.Int) ;
	Track803.DoneIN := EDGEPOS(S36Reed.In) ;
	Track804.DoneIN := EDGEPOS(S19Photo.Int) ;
	Track805.DoneIN := EDGENEG(S19Photo.Int) ;

	//TRACKINGSECTION END BLOCK CONDITIONS
	Tracking81.Blocks[9] := (Pause.Active) ;
	Tracking81.Blocks[10] := NOT(WashRun.In) ;
	Tracking81.Blocks[11] := NOT(FurnReady.Int) ;
	Tracking81.Blocks[12] := (S55Lever.In) ;
	Tracking81.ControlIN := Control.Achieved1 ;
	Tracking81.EMOStart := EMO.StartLatch ;
	Tracking81.ESClear := Control.ESClear ;
	Tracking81 ();
	Tracking81.ResMan := FALSE ;
	CASE Tracking81.Index OF
		0: //RESET ALL TRACKBIT FOR SELECTED TRACKINGSECTION
			Track811 := TrackClear ;
			Track812 := TrackClear ;
		1: //TRACK FROM S19Photo.Int (N) TO S21Photo.Int (P)
			Track812 := TrackClear ;
			//FB INPUTS
			Track811.FixedIN := Tracking81.FixedOUT ;
			Track811.Speed := Speeds.SpeedBatch ;
			Track811.TimeoutEN := TRUE ;
			Track811.TimeoutACK := Warn.Ack ;
			Track811.TimeoutBlock := (Warn.Block) ;
			Track811.DelayPT := TrackDelayPT.PTTrack811 ;
			//FB CALL
			Track811 ();
			//FB OUTPUTS
			CRE.o.Run[0] := Track811.RunOUT ;
			CLB.o.Run[0] := Track811.RunOUT ;
			CRE.Inv.Scale1.x := Track811.SpeedOUT ;
			CLB.Inv.Scale1.x := Track811.SpeedOUT ;
			IF(Track811.Done) THEN
				Tracking81.IndexIN := 2 ;
			END_IF
		2: //TRACK FROM S21Photo.Int (P) TO NOT(Tracking81.Blocked) (-)
			Track811 := TrackClear ;
			//FB INPUTS
			Track812.FixedIN := Tracking81.FixedOUT ;
			Track812.SolBlock := (S55Lever.In)OR NOT(WashRun.In) ;
			//FB CALL
			Track812 ();
			//FB OUTPUTS
			BatchAtExit.Auto := (Track812.SolOUT) ;
			IF(Track812.Done) THEN
				Tracking81.IndexIN := 0 ;
				Tracking82.IndexIN := 1 ;
			END_IF
	END_CASE

	//TRACKBIT DONE CONDITIONS
	Track811.DoneIN := EDGEPOS(S21Photo.Int) ;
	Track812.DoneIN := NOT(Tracking81.Blocked) ;

	//TRACKINGSECTION END BLOCK CONDITIONS
	Tracking82.ControlIN := Control.Achieved1 ;
	Tracking82.EMOStart := EMO.StartLatch ;
	Tracking82.ESClear := Control.ESClear ;
	Tracking82 ();
	Tracking82.ResMan := FALSE ;
	IF(CLB.LastSpeed = 0.0)THEN
		TrackDelayPT.PTTrack812 := 1000 ;
	ELSE
		TrackDelayPT.PTTrack812	:=	REAL_TO_UDINT((UDINT_TO_REAL(TrackDelayPT.PTTrack822)) *((10/CLB.LastSpeed)));
	END_IF
	CASE Tracking82.Index OF
		0: //RESET ALL TRACKBIT FOR SELECTED TRACKINGSECTION
			Track821 := TrackClear ;
			Track822 := TrackClear ;
		1: //TRACK FROM NOT(Tracking81.Blocked) (-) TO S21Photo.Int (N)
			Track822 := TrackClear ;
			//FB INPUTS
			Track821.FixedIN := Tracking82.FixedOUT ;
			Track821.Speed := Speeds.SpeedWash ;
			Track821.Analog := InvPerms.CLB.Analog ;
			Track821.SpeedAnalog := CLB.SpeedAnalog ;
			Track821.TimeoutEN := TRUE ;
			Track821.TimeoutACK := Warn.Ack ;
			Track821.TimeoutBlock := (Warn.Block) ;
			Track821.DelayPT := TrackDelayPT.PTTrack821 ;
			//FB CALL
			Track821 ();
			//FB OUTPUTS
			CLB.o.Run[0] := Track821.RunOUT ;
			CLB.Inv.Scale1.x := Track821.SpeedOUT ;
			WashStop.Auto := Track821.RunOUT ;
			BatchAtExit.Auto := (Track821.SolOUT) ;
			IF(Track821.Done) THEN
				Tracking82.IndexIN := 2 ;
			END_IF
		2: //TRACK FROM S21Photo.Int (N) TO Track821.DelayTON.Q (P)
			Track821 := TrackClear ;
			//FB INPUTS
			Track822.FixedIN := Tracking82.FixedOUT ;
			Track821.Speed := Speeds.SpeedWash ;
			Track821.Analog := InvPerms.CLB.Analog ;
			Track821.SpeedAnalog := CLB.SpeedAnalog ;
			Track822.TrackDelayEN := TRUE ;
			Track822.DelayPT := TrackDelayPT.PTTrack812 ;
			//FB CALL
			Track822 ();
			//FB OUTPUTS
			CLB.o.Run[0] := Track822.RunOUT ;
			CLB.Inv.Scale1.x := Track822.SpeedOUT ;
			WashStop.Auto := Track822.RunOUT ;
			BatchAtExit.Auto := (Track822.SolOUT) ;
			IF(Track822.Done) THEN
				Tracking82.IndexIN := 0 ;
			END_IF
	END_CASE

	//TRACKBIT DONE CONDITIONS
	Track821.DoneIN := EDGENEG(S21Photo.Int) ;

	//MANUAL BATCHING
	//TRACKINGSECTION END BLOCK CONDITIONS
	Tracking51.Blocks[1] := (Tracking70.Busy) ;
	Tracking51.Blocks[2] := (CLB.Input.Fault) ;
	Tracking51.Blocks[9] := (Pause.Active) ;
	Tracking51.Blocks[10] := NOT(WashRun.In) ;
	Tracking51.Blocks[11] := NOT(FurnReady.Int) ;
	Tracking51.Blocks[12] := (S55Lever.In) ;
	Tracking51.ControlIN := Control.Achieved1 ;
	Tracking51.EMOStart := EMO.StartLatch ;
	Tracking51.ESClear := Control.ESClear ;
	Tracking51 ();
	Tracking51.ResMan := FALSE ;
	IF(S58Lever.In) AND NOT((Tracking41.Busy) OR(Tracking50.Busy) OR(Tracking60.Busy) OR(Tracking70.Busy)) THEN
		S58Lever.Int := TRUE ;
	END_IF
	IF(S58Lever.Int)THEN
		Sol33Pal4.Auto := FALSE ;
	END_IF
	IF(S58Lever.Int) AND NOT(S58Lever.In) AND(Track511.Active)THEN
		IF EDGEPOS(S48Foot.In)THEN
			S58Lever.Int := FALSE ;
			Tracking51.IndexIN := 0 ;
		END_IF
	END_IF
	CASE Tracking51.Index OF
		0: //RESET ALL TRACKBIT FOR SELECTED TRACKINGSECTION
			Track511 := TrackClear ;
			Track512 := TrackClear ;
			Track513 := TrackClear ;
			//START CONDITION FOR LOADING
			IF(S58Lever.In) AND(S58Lever.Int)AND NOT((Tracking51.Busy) OR(Tracking70.Busy)) AND(Control.Achieved1)THEN
				Tracking51.IndexIN:=1;
			END_IF
			IF NOT(S58Lever.In)THEN
				S58Lever.Int := FALSE ;
			END_IF
		1: //TRACK FROM S58Lever.Int (P) TO S66PB.In (P)
			Track512 := TrackClear ;
			Track513 := TrackClear ;
			//FB INPUTS
			Track511.FixedIN := Tracking51.FixedOUT ;
			Track511.Speed := Speeds.SpeedEntry ;
			Track511.RunBlock := NOT(S48Foot.In) OR (S20Photo.Int) ;
			//FB CALL
			Track511 ();
			//FB OUTPUTS
			CRE.o.Run[0] := Track511.RunOUT ;
			CRE.Inv.Scale1.x := Track511.SpeedOUT ;
			CLB.o.Run[0] := Track511.RunOUT ;
			CLB.Inv.Scale1.x := Track511.SpeedOUT ;
			IF(Track511.Done)THEN
				Tracking51.IndexIN := 2 ;
			END_IF
		2: //TRACK FROM S66PB.In (P) TO S21Photo.Int (P)
			Track511 := TrackClear ;
			Track513 := TrackClear ;
			//FB INPUTS
			Track512.FixedIN := Tracking51.FixedOUT ;
			Track512.Speed := Speeds.SpeedBatch ;
			Track512.TimeoutEN := TRUE ;
			Track512.TimeoutACK := Warn.Ack ;
			Track512.TimeoutBlock := (Warn.Block) ;
			Track512.DelayPT := TrackDelayPT.PTTrack603 ;
			//FB CALL
			Track512 ();
			//FB OUTPUTS
			CRE.o.Run[0] := Track512.RunOUT ;
			CRE.Inv.Scale1.x := Track512.SpeedOUT ;
			CLB.o.Run[0] := Track512.RunOUT ;
			CLB.Inv.Scale1.x := Track512.SpeedOUT ;
			IF(Track512.Done)THEN
				Tracking51.IndexIN := 3 ;
			END_IF
		3: //TRACK FROM S21Photo.Int (P) TO NOT(Tracking51.Blocked) (-)
			Track511 := TrackClear ;
			Track512 := TrackClear ;
			//FB INPUTS
			Track513.FixedIN := Tracking51.FixedOUT ;
			//FB CALL
			Track513 ();
			//FB OUTPUTS
			IF(Track513.Done) THEN
				Tracking51.IndexIN := 0 ;
				Tracking70.IndexIN := 1 ;
			END_IF
	END_CASE

	//TRACKBIT DONE CONDITIONS
	Track511.DoneIN := EDGEPOS(S66PB.In) ;
	Track512.DoneIN := EDGEPOS(S21Photo.Int) ;
	Track513.DoneIN := NOT(Tracking51.Blocked) ;

END_PROGRAM
```

### Program Logical/Automatic/FlipUpArms (IEC)

#### Cyclic.st
```iecst
PROGRAM _CYCLIC

	//------------------------------------------------------
	//FLIP UP ARMS FASTMAXX 1
	//FB INPUTS
	ArmsTemp1.Down[1] := S100Reed.In ;
	ArmsTemp1.Down[2] := S102Reed.In ;
	ArmsTemp1.Down[3] := S104Reed.In ;
	ArmsTemp1.Down[4] := S106Reed.In ;
	ArmsTemp1.Down[5] := S108Reed.In ;
	ArmsTemp1.Down[6] := S110Reed.In ;
	ArmsTemp1.Down[7] := S112Reed.In ;
	ArmsTemp1.Down[8] := S114Reed.In ;
	ArmsTemp1.Up[1] := S101Reed.In ;
	ArmsTemp1.Up[2] := S103Reed.In ;
	ArmsTemp1.Up[3] := S105Reed.In ;
	ArmsTemp1.Up[4] := S107Reed.In ;
	ArmsTemp1.Up[5] := S109Reed.In ;
	ArmsTemp1.Up[6] := S111Reed.In ;
	ArmsTemp1.Up[7] := S113Reed.In ;
	ArmsTemp1.Up[8] := S115Reed.In ;
	ArmsTemp1.Arms := 4 ;
	ArmsTemp1.Raise := Ax1.RaiseArms ;
	ArmsTemp1.HiVol := Ax1.HiVol ;
	ArmsTemp1.ArmPos := ArmsPerm1.Position ;
	//CALL FB
	ArmsTemp1 ();
	//FB OUTPUTS
	Sol5Arm1.Auto := ArmsTemp1.OUT[1] ;
	Sol6Arm2.Auto := ArmsTemp1.OUT[2] ;
	Sol7Arm3.Auto := ArmsTemp1.OUT[3] ;
	Sol8Arm4.Auto := ArmsTemp1.OUT[4] ;

	//FLIP UP ARMS FASTMAXX 2
	//FB INPUTS
	ArmsTemp2.Down[1] := S120Reed.In ;
	ArmsTemp2.Down[2] := S122Reed.In ;
	ArmsTemp2.Down[3] := S124Reed.In ;
	ArmsTemp2.Down[4] := S126Reed.In ;
	ArmsTemp2.Up[1] := S121Reed.In ;
	ArmsTemp2.Up[2] := S123Reed.In ;
	ArmsTemp2.Up[3] := S125Reed.In ;
	ArmsTemp2.Up[4] := S127Reed.In ;
	ArmsTemp2.Arms := 2 ;
	ArmsTemp2.Raise := Ax2.RaiseArms ;
	ArmsTemp2.HiVol := Ax2.HiVol ;
	ArmsTemp2.ArmPos := ArmsPerm2.Position ;
	//CALL FB
	ArmsTemp2 ();
	//FB OUTPUTS
	Sol14Arm6.Auto := ArmsTemp2.OUT[1] ;
	Sol15Arm7.Auto := ArmsTemp2.OUT[2] ;

END_PROGRAM
```

### Program Logical/Automatic/Outputs (IEC) - Set outputs from array conditions

#### OutputsCyclic.st - Cyclic code
```iecst
(********************************************************************
 * COPYRIGHT --
 ********************************************************************
 * Program: Outputs
 * File: OutputsCyclic.st
 ********************************************************************
 * Implementation of program Outputs
 ********************************************************************)

PROGRAM _CYCLIC

    //INDIVIDUAL LEG TEST CONTROL
	CASE LegTest.Index OF
		TEST_OFF:
			LegTest.Index := LIMIT(TEST_OFF,LegTest.Index, TEST_ON_STOP) ;
			LegTest.Disp := HIDE ;
		TEST_ON_STOP:
			LegTest.Index := LIMIT(TEST_OFF,LegTest.Index, TEST_LEG4) ;
			CL1.Inv.Test := 0 ;
			CS1.Inv.Test := 0 ;
			CV1.Inv.Test := 0 ;
			CC1.Inv.Test := 0 ;
			CC2.Inv.Test := 0 ;
			CS2.Inv.Test := 0 ;
			CV2.Inv.Test := 0 ;
			CC3.Inv.Test := 0 ;
			CC4.Inv.Test := 0 ;
			CB1.Inv.Test := 0 ;
			CB2.Inv.Test := 0 ;
			CRB.Inv.Test := 0 ;
			CRE.Inv.Test := 0 ;
			CLB.Inv.Test := 0 ;
			LegTest.Disp := SHOW ;
		TEST_LEG1:
			CL1.Inv.Test := 4 ;
			CS1.Inv.Test := 4 ;
			CV1.Inv.Test := 4 ;
			CC1.Inv.Test := 4 ;
			LegTest.Disp := SHOW ;
		TEST_LEG2:
			CC2.Inv.Test := 4 ;
			CS2.Inv.Test := 4 ;
			CV2.Inv.Test := 4 ;
			CC3.Inv.Test := 4 ;
			LegTest.Disp := SHOW ;
		TEST_LEG3:
			CC4.Inv.Test := 4 ;
			CB1.Inv.Test := 4 ;
			CB2.Inv.Test := 4 ;
			CRB.Inv.Test := 4 ;
			LegTest.Disp := SHOW ;
		TEST_LEG4:
			CASE InvPerms.CRE.Analog OF
				NO_ANALOG:
					CRE.Inv.Test := 4 ;
					CLB.Inv.Test := 4 ;
				ELSE
					CRE.Inv.Test := 14 ;
					CLB.Inv.Test := 14 ;
			END_CASE
			LegTest.Disp := SHOW ;
	END_CASE

	//CONVEYOR TEST MODES
	//FB INPUTS
	CL1Test.SpeedIN := Speeds ;
	CL1Test.TestSpeedIN := CL1.Inv.SpeedTest ;
	CL1Test.Index := CL1.Inv.Test ;
	CL1Test.AutoSpeedIN := CL1.Inv.Scale1.x ;
	//CALL FB
	CL1Test ();
	//FB OUTPUTS
	CL1.o.Run[3] := CL1Test.Run ;
	CL1.o.Rev[3] := CL1Test.Rev ;
	CL1.Inv.Scale1.x := CL1Test.Speed ;

	//FB INPUTS
	CS1Test.SpeedIN := Speeds ;
	CS1Test.TestSpeedIN := CS1.Inv.SpeedTest ;
	CS1Test.Index := CS1.Inv.Test ;
	CS1Test.AutoSpeedIN := CS1.Inv.Scale1.x ;
	//CALL FB
	CS1Test ();
	//FB OUTPUTS
	CS1.o.Run[3] := CS1Test.Run ;
	CS1.o.Rev[3] := CS1Test.Rev ;
	CS1.Inv.Scale1.x := CS1Test.Speed ;

	//FB INPUTS
	CV1Test.SpeedIN := Speeds ;
	CV1Test.TestSpeedIN := CV1.Inv.SpeedTest ;
	CV1Test.Index := CV1.Inv.Test ;
	CV1Test.AutoSpeedIN := CV1.Inv.Scale1.x ;
	//CALL FB
	CV1Test ();
	//FB OUTPUTS
	CV1.o.Run[3] := CV1Test.Run ;
	CV1.o.Rev[3] := CV1Test.Rev ;
	CV1.Inv.Scale1.x := CV1Test.Speed ;

	//FB INPUTS
	CC1Test.SpeedIN := Speeds ;
	CC1Test.TestSpeedIN := CC1.Inv.SpeedTest ;
	CC1Test.Index := CC1.Inv.Test ;
	CC1Test.AutoSpeedIN := CC1.Inv.Scale1.x ;
	//CALL FB
	CC1Test ();
	//FB OUTPUTS
	CC1.o.Run[3] := CC1Test.Run ;
	CC1.o.Rev[3] := CC1Test.Rev ;
	CC1.Inv.Scale1.x := CC1Test.Speed ;

	//FB INPUTS
	CC2Test.SpeedIN := Speeds ;
	CC2Test.TestSpeedIN := CC2.Inv.SpeedTest ;
	CC2Test.Index := CC2.Inv.Test ;
	CC2Test.AutoSpeedIN := CC2.Inv.Scale1.x ;
	//CALL FB
	CC2Test ();
	//FB OUTPUTS
	CC2.o.Run[3] := CC2Test.Run ;
	CC2.o.Rev[3] := CC2Test.Rev ;
	CC2.Inv.Scale1.x := CC2Test.Speed ;

	//FB INPUTS
	CS2Test.SpeedIN := Speeds ;
	CS2Test.TestSpeedIN := CS2.Inv.SpeedTest ;
	CS2Test.Index := CS2.Inv.Test ;
	CS2Test.AutoSpeedIN := CS2.Inv.Scale1.x ;
	//CALL FB
	CS2Test ();
	//FB OUTPUTS
	CS2.o.Run[3] := CS2Test.Run ;
	CS2.o.Rev[3] := CS2Test.Rev ;
	CS2.Inv.Scale1.x := CS2Test.Speed ;

	//FB INPUTS
	CV2Test.SpeedIN := Speeds ;
	CV2Test.TestSpeedIN := CV2.Inv.SpeedTest ;
	CV2Test.Index := CV2.Inv.Test ;
	CV2Test.AutoSpeedIN := CV2.Inv.Scale1.x ;
	//CALL FB
	CV2Test ();
	//FB OUTPUTS
	CV2.o.Run[3] := CV2Test.Run ;
	CV2.o.Rev[3] := CV2Test.Rev ;
	CV2.Inv.Scale1.x := CV2Test.Speed ;

	//FB INPUTS
	CC3Test.SpeedIN := Speeds ;
	CC3Test.TestSpeedIN := CC3.Inv.SpeedTest ;
	CC3Test.Index := CC3.Inv.Test ;
	CC3Test.AutoSpeedIN := CC3.Inv.Scale1.x ;
	//CALL FB
	CC3Test ();
	//FB OUTPUTS
	CC3.o.Run[3] := CC3Test.Run ;
	CC3.o.Rev[3] := CC3Test.Rev ;
	CC3.Inv.Scale1.x := CC3Test.Speed ;

	//FB INPUTS
	CC4Test.SpeedIN := Speeds ;
	CC4Test.TestSpeedIN := CC4.Inv.SpeedTest ;
	CC4Test.Index := CC4.Inv.Test ;
	CC4Test.AutoSpeedIN := CC4.Inv.Scale1.x ;
	//CALL FB
	CC4Test ();
	//FB OUTPUTS
	CC4.o.Run[3] := CC4Test.Run ;
	CC4.o.Rev[3] := CC4Test.Rev ;
	CC4.Inv.Scale1.x := CC4Test.Speed ;

	//FB INPUTS
	CB1Test.SpeedIN := Speeds ;
	CB1Test.TestSpeedIN := CB1.Inv.SpeedTest ;
	CB1Test.Index := CB1.Inv.Test ;
	CB1Test.AutoSpeedIN := CB1.Inv.Scale1.x ;
	//CALL FB
	CB1Test ();
	//FB OUTPUTS
	CB1.o.Run[3] := CB1Test.Run ;
	CB1.o.Rev[3] := CB1Test.Rev ;
	CB1.Inv.Scale1.x := CB1Test.Speed ;

	//FB INPUTS
	CB2Test.SpeedIN := Speeds ;
	CB2Test.TestSpeedIN := CB2.Inv.SpeedTest ;
	CB2Test.Index := CB2.Inv.Test ;
	CB2Test.AutoSpeedIN := CB2.Inv.Scale1.x ;
	//CALL FB
	CB2Test ();
	//FB OUTPUTS
	CB2.o.Run[3] := CB2Test.Run ;
	CB2.o.Rev[3] := CB2Test.Rev ;
	CB2.Inv.Scale1.x := CB2Test.Speed ;

	//FB INPUTS
	CRBTest.SpeedIN := Speeds ;
	CRBTest.TestSpeedIN := CRB.Inv.SpeedTest ;
	CRBTest.Index := CRB.Inv.Test ;
	CRBTest.AutoSpeedIN := CRB.Inv.Scale1.x ;
	//CALL FB
	CRBTest ();
	//FB OUTPUTS
	CRB.o.Run[3] := CRBTest.Run ;
	CRB.o.Rev[3] := CRBTest.Rev ;
	CRB.Inv.Scale1.x := CRBTest.Speed ;

	//FB INPUTS
	CRETest.SpeedIN := Speeds ;
	CRETest.TestSpeedIN := CRE.Inv.SpeedTest ;
	CRETest.Index := CRE.Inv.Test ;
	CRETest.AutoSpeedIN := CRE.Inv.Scale1.x ;
	//CALL FB
	CRETest ();
	//FB OUTPUTS
	CRE.o.Run[3] := CRETest.Run ;
	CRE.o.Rev[3] := CRETest.Rev ;
	CRE.Inv.Scale1.x := CRETest.Speed ;

	//FB INPUTS
	CLBTest.SpeedIN := Speeds ;
	CLBTest.TestSpeedIN := CLB.Inv.SpeedTest ;
	CLBTest.AnalogSpeedIN := CLB.SpeedAnalog ;
	CLBTest.Index := CLB.Inv.Test ;
	CLBTest.AutoSpeedIN := CLB.Inv.Scale1.x ;
	//CALL FB
	CLBTest ();
	//FB OUTPUTS
	CLB.o.Run[3] := CLBTest.Run ;
	CLB.o.Rev[3] := CLBTest.Rev ;
	CLB.Inv.Scale1.x := CLBTest.Speed ;

	//------------------------------------------------------
	//CONVEYOR CONTROL
	IF NOT(Control.Test) THEN
		IF NOT(Control.Achieved1) OR(Control.ESClear) THEN
			FOR i:= 0 TO 5 DO
				CL1.o.Run[i]   :=  FALSE   ;
				CL1.o.Rev[i]   :=  FALSE   ;
				CS1.o.Run[i]   :=  FALSE   ;
				CS1.o.Rev[i]   :=  FALSE   ;
				CV1.o.Run[i]   :=  FALSE   ;
				CV1.o.Rev[i]   :=  FALSE   ;
				CC1.o.Run[i]   :=  FALSE   ;
				CC1.o.Rev[i]   :=  FALSE   ;
				CC2.o.Run[i]   :=  FALSE   ;
				CC2.o.Rev[i]   :=  FALSE   ;
				CS2.o.Run[i]   :=  FALSE   ;
				CS2.o.Rev[i]   :=  FALSE   ;
				CV2.o.Run[i]   :=  FALSE   ;
				CV2.o.Rev[i]   :=  FALSE   ;
				CC3.o.Run[i]   :=  FALSE   ;
				CC3.o.Rev[i]   :=  FALSE   ;
				CC4.o.Run[i]   :=  FALSE   ;
				CC4.o.Rev[i]   :=  FALSE   ;
				CB1.o.Run[i]   :=  FALSE   ;
				CB1.o.Rev[i]   :=  FALSE   ;
				CB2.o.Run[i]   :=  FALSE   ;
				CB2.o.Rev[i]   :=  FALSE   ;
				CRB.o.Run[i]   :=  FALSE   ;
				CRB.o.Rev[i]   :=  FALSE   ;
				CRE.o.Run[i]   :=  FALSE   ;
				CRE.o.Rev[i]   :=  FALSE   ;
				CLB.o.Run[i]   :=  FALSE   ;
				CLB.o.Rev[i]   :=  FALSE   ;
			END_FOR
		END_IF
	END_IF

	FOR i:= 0 TO 5 DO
		IF CL1.o.Run[i] = TRUE THEN
			CL1.Output.CMDD_03 :=  TRUE    ;
			EXIT;
		ELSE
			CL1.Output.CMDD_03 :=  FALSE   ;
		END_IF
	END_FOR

	FOR i:= 0 TO 5 DO
		IF CL1.o.Rev[i] = TRUE THEN
			CL1.Output.CMDD_03 :=  TRUE   ;
			CL1.Output.CMDD_11 :=  TRUE    ;
			EXIT;
		ELSE
			CL1.Output.CMDD_11 :=  FALSE   ;
		END_IF
	END_FOR

	FOR i:= 0 TO 5 DO
		IF CS1.o.Run[i] = TRUE THEN
			CS1.Output.CMDD_03 :=  TRUE    ;
			EXIT;
		ELSE
			CS1.Output.CMDD_03 :=  FALSE   ;
		END_IF
	END_FOR

	FOR i:= 0 TO 5 DO
		IF CS1.o.Rev[i] = TRUE THEN
			CS1.Output.CMDD_03 :=  TRUE   ;
			CS1.Output.CMDD_11 :=  TRUE    ;
			EXIT;
		ELSE
			CS1.Output.CMDD_11 :=  FALSE   ;
		END_IF
	END_FOR

	FOR i:= 0 TO 5 DO
		IF CV1.o.Run[i] = TRUE THEN
			CV1.Output.CMDD_03 :=  TRUE    ;
			EXIT;
		ELSE
			CV1.Output.CMDD_03 :=  FALSE   ;
		END_IF
	END_FOR

	FOR i:= 0 TO 5 DO
		IF CV1.o.Rev[i] = TRUE THEN
			CV1.Output.CMDD_03 :=  TRUE   ;
			CV1.Output.CMDD_11 :=  TRUE    ;
			EXIT;
		ELSE
			CV1.Output.CMDD_11 :=  FALSE   ;
		END_IF
	END_FOR

	FOR i:= 0 TO 5 DO
		IF CC1.o.Run[i] = TRUE THEN
			CC1.Output.CMDD_03 :=  TRUE    ;
			EXIT;
		ELSE
			CC1.Output.CMDD_03 :=  FALSE   ;
		END_IF
	END_FOR

	FOR i:= 0 TO 5 DO
		IF CC1.o.Rev[i] = TRUE THEN
			CC1.Output.CMDD_03 :=  TRUE   ;
			CC1.Output.CMDD_11 :=  TRUE    ;
			EXIT;
		ELSE
			CC1.Output.CMDD_11 :=  FALSE   ;
		END_IF
	END_FOR

	FOR i:= 0 TO 5 DO
		IF CC2.o.Run[i] = TRUE THEN
			CC2.Output.CMDD_03 :=  TRUE    ;
			EXIT;
		ELSE
			CC2.Output.CMDD_03 :=  FALSE   ;
		END_IF
	END_FOR

	FOR i:= 0 TO 5 DO
		IF CC2.o.Rev[i] = TRUE THEN
			CC2.Output.CMDD_03 :=  TRUE   ;
			CC2.Output.CMDD_11 :=  TRUE    ;
			EXIT;
		ELSE
			CC2.Output.CMDD_11 :=  FALSE   ;
		END_IF
	END_FOR

	FOR i:= 0 TO 5 DO
		IF CS2.o.Run[i] = TRUE THEN
			CS2.Output.CMDD_03 :=  TRUE    ;
			EXIT;
		ELSE
			CS2.Output.CMDD_03 :=  FALSE   ;
		END_IF
	END_FOR

	FOR i:= 0 TO 5 DO
		IF CS2.o.Rev[i] = TRUE THEN
			CS2.Output.CMDD_03 :=  TRUE   ;
			CS2.Output.CMDD_11 :=  TRUE    ;
			EXIT;
		ELSE
			CS2.Output.CMDD_11 :=  FALSE   ;
		END_IF
	END_FOR

	FOR i:= 0 TO 5 DO
		IF CV2.o.Run[i] = TRUE THEN
			CV2.Output.CMDD_03 :=  TRUE    ;
			EXIT;
		ELSE
			CV2.Output.CMDD_03 :=  FALSE   ;
		END_IF
	END_FOR

	FOR i:= 0 TO 5 DO
		IF CV2.o.Rev[i] = TRUE THEN
			CV2.Output.CMDD_03 :=  TRUE   ;
			CV2.Output.CMDD_11 :=  TRUE    ;
			EXIT;
		ELSE
			CV2.Output.CMDD_11 :=  FALSE   ;
		END_IF
	END_FOR

	FOR i:= 0 TO 5 DO
		IF CC3.o.Run[i] = TRUE THEN
			CC3.Output.CMDD_03 :=  TRUE    ;
			EXIT;
		ELSE
			CC3.Output.CMDD_03 :=  FALSE   ;
		END_IF
	END_FOR

	FOR i:= 0 TO 5 DO
		IF CC3.o.Rev[i] = TRUE THEN
			CC3.Output.CMDD_03 :=  TRUE   ;
			CC3.Output.CMDD_11 :=  TRUE    ;
			EXIT;
		ELSE
			CC3.Output.CMDD_11 :=  FALSE   ;
		END_IF
	END_FOR

	FOR i:= 0 TO 5 DO
		IF CC4.o.Run[i] = TRUE THEN
			CC4.Output.CMDD_03 :=  TRUE    ;
			EXIT;
		ELSE
			CC4.Output.CMDD_03 :=  FALSE   ;
		END_IF
	END_FOR

	FOR i:= 0 TO 5 DO
		IF CC4.o.Rev[i] = TRUE THEN
			CC4.Output.CMDD_03 :=  TRUE   ;
			CC4.Output.CMDD_11 :=  TRUE    ;
			EXIT;
		ELSE
			CC4.Output.CMDD_11 :=  FALSE   ;
		END_IF
	END_FOR

	FOR i:= 0 TO 5 DO
		IF CB1.o.Run[i] = TRUE THEN
			CB1.Output.CMDD_03 :=  TRUE    ;
			EXIT;
		ELSE
			CB1.Output.CMDD_03 :=  FALSE   ;
		END_IF
	END_FOR

	FOR i:= 0 TO 5 DO
		IF CB1.o.Rev[i] = TRUE THEN
			CB1.Output.CMDD_03 :=  TRUE   ;
			CB1.Output.CMDD_11 :=  TRUE    ;
			EXIT;
		ELSE
			CB1.Output.CMDD_11 :=  FALSE   ;
		END_IF
	END_FOR

	FOR i:= 0 TO 5 DO
		IF CB2.o.Run[i] = TRUE THEN
			CB2.Output.CMDD_03 :=  TRUE    ;
			EXIT;
		ELSE
			CB2.Output.CMDD_03 :=  FALSE   ;
		END_IF
	END_FOR

	FOR i:= 0 TO 5 DO
		IF CB2.o.Rev[i] = TRUE THEN
			CB2.Output.CMDD_03 :=  TRUE   ;
			CB2.Output.CMDD_11 :=  TRUE    ;
			EXIT;
		ELSE
			CB2.Output.CMDD_11 :=  FALSE   ;
		END_IF
	END_FOR

	FOR i:= 0 TO 5 DO
		IF CRB.o.Run[i] = TRUE THEN
			CRB.Output.CMDD_03 :=  TRUE    ;
			EXIT;
		ELSE
			CRB.Output.CMDD_03 :=  FALSE   ;
		END_IF
	END_FOR

	FOR i:= 0 TO 5 DO
		IF CRB.o.Rev[i] = TRUE THEN
			CRB.Output.CMDD_03 :=  TRUE   ;
			CRB.Output.CMDD_11 :=  TRUE    ;
			EXIT;
		ELSE
			CRB.Output.CMDD_11 :=  FALSE   ;
		END_IF
	END_FOR

	FOR i:= 0 TO 5 DO
		IF CRE.o.Run[i] = TRUE THEN
			CRE.Output.CMDD_03 :=  TRUE    ;
			EXIT;
		ELSE
			CRE.Output.CMDD_03 :=  FALSE   ;
		END_IF
	END_FOR

	FOR i:= 0 TO 5 DO
		IF CRE.o.Rev[i] = TRUE THEN
			CRE.Output.CMDD_03 :=  TRUE   ;
			CRE.Output.CMDD_11 :=  TRUE    ;
			EXIT;
		ELSE
			CRE.Output.CMDD_11 :=  FALSE   ;
		END_IF
	END_FOR

	FOR i:= 0 TO 5 DO
		IF CLB.o.Run[i] = TRUE THEN
			CLB.Output.CMDD_03 :=  TRUE    ;
			CLB.LastSpeed := (CLB.o.SpeedRef/10) * (ScalePerm.CLBScale/50) ;
			EXIT;
		ELSE
			CLB.Output.CMDD_03 :=  FALSE   ;
		END_IF
	END_FOR

	FOR i:= 0 TO 5 DO
		IF CLB.o.Rev[i] = TRUE THEN
			CLB.Output.CMDD_03 :=  TRUE   ;
			CLB.Output.CMDD_11 :=  TRUE    ;
			EXIT;
		ELSE
			CLB.Output.CMDD_11 :=  FALSE   ;
		END_IF
	END_FOR

END_PROGRAM
```

### Package Logical/Motion - A package of related programs and data objects.

### Motion1.var
```iecst
(********************************************************************
 * COPYRIGHT --
 ********************************************************************
 * Package: Motion1
 * File: Motion1.var
 * Author: nicke
 * Created: February, 2012
 ********************************************************************
 * Variables of package Motion1
 ********************************************************************)
VAR
	ErrorACKs2 : ARRAY[0..5] OF BOOL := [6(FALSE)];
	ScreenACK2 : BOOL := FALSE;
	ScreenACK1 : BOOL := FALSE;
	ErrorACKs1 : ARRAY[0..5] OF BOOL := [6(FALSE)];
	Axis1DigiIPsFromX67 : AxisSwitchCfg;
	Axis1StatusBitsCyclicRead : MC_BR_InitCyclicRead;
	Axis2DigiIPsFromX67 : AxisSwitchCfg;
	Axis2StatusBitsCyclicRead : MC_BR_InitCyclicRead;
	machine : Machine;
	machine2 : Machine;
	MC_Home_0 : MC_Home;
	MC_Home_2 : MC_Home;
	MC_MoveAbsolute_0 : MC_MoveAbsolute;
	MC_MoveAbsolute_2 : MC_MoveAbsolute;
	MC_MoveVelocity_0 : MC_MoveVelocity;
	MC_MoveVelocity_1 : MC_MoveVelocity;
	MC_MoveVelocity_3 : MC_MoveVelocity;
	MC_MoveVelocity_2 : MC_MoveVelocity;
	MC_Power_0 : MC_Power;
	MC_Power_2 : MC_Power;
	MC_ReadActualPosition_0 : MC_ReadActualPosition;
	MC_ReadActualPosition_2 : MC_ReadActualPosition;
	MC_ReadActualVelocity_0 : MC_ReadActualVelocity;
	MC_ReadActualVelocity_2 : MC_ReadActualVelocity;
	MC_ReadAxisError_0 : MC_ReadAxisError;
	MC_ReadAxisError_2 : MC_ReadAxisError;
	MC_ReadStatus_0 : MC_ReadStatus;
	MC_ReadStatus_2 : MC_ReadStatus;
	MC_Reset_0 : MC_Reset;
	MC_Reset_2 : MC_Reset;
	MC_Stop_0 : MC_Stop;
	MC_Stop_2 : MC_Stop;
END_VAR
```

### Data object Logical/Motion/english (Ett) - ACP10: ErrorText data object.

- english.ett (not shown)

### Data object Logical/Motion/table_par1 (Apt) - ACOPOS Parameter Table

#### table_par1.apt
```
AcoposParameterTable:
  Root Parameters:
    M1 (Disabled=TRUE, StructureEdit=FALSE)  // 8LSA45.E2030D000-0 Rev.C3
      General parameters (Disabled=TRUE)
        30 = 0x0002 (Name=MOTOR_TYPE, Disabled=TRUE)  // Motor: Type
        31 = 0x0203 (Name=MOTOR_COMPATIBILITY, Disabled=TRUE)  // Motor: Software compatibility
        46 = 1 (Name=MOTOR_WIND_CONNECT, Disabled=TRUE)  // Motor: Winding connection
        47 = 5 (Name=MOTOR_POLEPAIRS, Disabled=TRUE)  // Motor: Number of pole-pairs
      Brake parameters (Disabled=TRUE)
        42 = 0 (Name=MOTOR_BRAKE_CURR_RATED, Unit=A, Disabled=TRUE)  // Motor holding brake: Rated current
        43 = 0 (Name=MOTOR_BRAKE_TORQ_RATED, Unit=Nm, Disabled=TRUE)  // Motor holding brake: Rated torque
        44 = 0 (Name=MOTOR_BRAKE_ON_TIME, Unit=s, Disabled=TRUE)  // Motor holding brake: Engaging delay
        45 = 0 (Name=MOTOR_BRAKE_OFF_TIME, Unit=s, Disabled=TRUE)  // Motor holding brake: Release delay
      Thermo sensor parameters (Disabled=TRUE)
        64 = 632 (Name=MOTOR_TEMPSENS_PAR1, Disabled=TRUE)  // Temperature sensor: Parameter 1
        65 = 2225 (Name=MOTOR_TEMPSENS_PAR2, Disabled=TRUE)  // Temperature sensor: Parameter 2
        66 = -30 (Name=MOTOR_TEMPSENS_PAR3, Disabled=TRUE)  // Temperature sensor: Parameter 3
        67 = 5.7266 (Name=MOTOR_TEMPSENS_PAR4, Disabled=TRUE)  // Temperature sensor: Parameter 4
        68 = 36.0938 (Name=MOTOR_TEMPSENS_PAR5, Disabled=TRUE)  // Temperature sensor: Parameter 5
        69 = 62.9375 (Name=MOTOR_TEMPSENS_PAR6, Disabled=TRUE)  // Temperature sensor: Parameter 6
        70 = 87.25 (Name=MOTOR_TEMPSENS_PAR7, Disabled=TRUE)  // Temperature sensor: Parameter 7
        71 = 109.6016 (Name=MOTOR_TEMPSENS_PAR8, Disabled=TRUE)  // Temperature sensor: Parameter 8
        72 = 130.3984 (Name=MOTOR_TEMPSENS_PAR9, Disabled=TRUE)  // Temperature sensor: Parameter 9
        73 = 150 (Name=MOTOR_TEMPSENS_PAR10, Disabled=TRUE)  // Temperature sensor: Parameter 10
        75 = 0 (Name=MOTOR_THERMAL_CONST, Unit=s, Disabled=TRUE)  // Motor: Thermal time constant (for MOTOR_COMPATIBILITY 0x0202)
      Motor parameters (Disabled=TRUE)
        48 = 400 (Name=MOTOR_VOLTAGE_RATED, Unit=V, Disabled=TRUE)  // Motor: Rated voltage
        49 = 98.43 (Name=MOTOR_VOLTAGE_CONST, Unit=mV*min, Disabled=TRUE)  // Motor: Voltage constant
        50 = 3000 (Name=MOTOR_SPEED_RATED, Unit=1/min, Disabled=TRUE)  // Motor: Rated speed
        51 = 12000 (Name=MOTOR_SPEED_MAX, Unit=1/min, Disabled=TRUE)  // Motor: Maximum speed
        52 = 8 (Name=MOTOR_TORQ_STALL, Unit=Nm, Disabled=TRUE)  // Motor: Stall torque
        53 = 6.16 (Name=MOTOR_TORQ_RATED, Unit=Nm, Disabled=TRUE)  // Motor: Rated torque
        54 = 30.4 (Name=MOTOR_TORQ_MAX, Unit=Nm, Disabled=TRUE)  // Motor: Peak torque
        55 = 1.628 (Name=MOTOR_TORQ_CONST, Unit=Nm/A, Disabled=TRUE)  // Motor: Torque constant
        56 = 4.913619 (Name=MOTOR_CURR_STALL, Unit=A, Disabled=TRUE)  // Motor: Stall current
        57 = 3.783487 (Name=MOTOR_CURR_RATED, Unit=A, Disabled=TRUE)  // Motor: Rated current
        58 = 29.174615 (Name=MOTOR_CURR_MAX, Unit=A, Disabled=TRUE)  // Motor: Peak current
        59 = 0.6362 (Name=MOTOR_WIND_CROSS_SECT, Unit=mm², Disabled=TRUE)  // Motor: Line cross section
        60 = 2.4891 (Name=MOTOR_STATOR_RESISTANCE, Unit=Ohm, Disabled=TRUE)  // Motor: Stator resistance
        61 = 0.021797 (Name=MOTOR_STATOR_INDUCTANCE, Unit=Henry, Disabled=TRUE)  // Motor: Stator inductance
        62 = 0.000358 (Name=MOTOR_INERTIA, Unit=kgm², Disabled=TRUE)  // Motor: Moment of inertia
        63 = 1e+006 (Name=MOTOR_COMMUT_OFFSET, Unit=rad, Disabled=TRUE)  // Motor: Commutation offset
        849 = 2100 (Name=MOTOR_TAU_THERM, Unit=s, Disabled=TRUE)  // Motor: Thermal time constant
      Isolation parameters (Disabled=TRUE)
        74 = 110 (Name=MOTOR_WIND_TEMP_MAX, Unit=°C, Disabled=TRUE)  // Temperature sensor: Limit temperature
    SS2 (StructureEdit=FALSE)  // 8AC120.00
      97 = ncENDAT (Name=ENCOD_TYPE)  // Encoder1: Type
```

### Data object Logical/Motion/axis1 (Ax) - ACP10: Axis data object.

#### axis1.ax
```
InitParameter (Version=2.50.1, NcSwId=ACP10)
  ACP10AXIS_typ:
    dig_in:
      level:
        reference = ncACTIV_HI
        pos_hw_end = ncACTIV_LO
        neg_hw_end = ncACTIV_LO
        trigger1 = ncACTIV_HI
        trigger2 = ncACTIV_HI
    encoder_if:
      parameter:
        count_dir = ncINVERSE
        scaling:
          load:
            units = 1449275
            rev_motor = 10000
    limit:
      parameter:
        v_pos = 10000
        v_neg = 10000
        a1_pos = 50000
        a2_pos = 50000
        a1_neg = 50000
        a2_neg = 50000
        t_jolt = 0.1
        t_in_pos = 0
        pos_sw_end = 8388607
        neg_sw_end = -8388608
        ds_warning = 500
        ds_stop = 1000
        a_stop = 1e+030
        dv_stop = 0
        dv_stop_mode = ncOFF
    controller:
      mode = ncPOSITION
      position:
        kv = 340.0
        tn = 0
        t_predict = 0.0004
        t_total = 0.0004
        p_max = 1e+030
        i_max = 0
      speed:
        kv = 0.6
        tn = 0
        t_filter = 0.0008
        isq_filter1:
          type = ncOFF
          a0 = 0
          a1 = 0
          b0 = 0
          b1 = 0
          b2 = 0
          c0_par_id = 0
          c1_par_id = 0
        isq_filter2:
          type = ncOFF
          a0 = 0
          a1 = 0
          b0 = 0
          b1 = 0
          b2 = 0
          c0_par_id = 0
          c1_par_id = 0
        isq_filter3:
          type = ncOFF
          a0 = 0
          a1 = 0
          b0 = 0
          b1 = 0
          b2 = 0
          c0_par_id = 0
          c1_par_id = 0
      uf:
        type = ncLINEAR
        auto_config = ncMOTOR_PAR
        u0 = 0
        un = 0
        fn = 50
        k_f_slip = 0
      ff:
        torque_load = 0
        torque_pos = 1.19512
        torque_neg = 1.2393
        kv_torque = 0.565411
        inertia = 0.00760164
        t_filter_a = 0
    move:
      stop:
        parameter[0]:
          decel_ramp = ncA_LIMIT
          controller = ncON
        parameter[1]:
          decel_ramp = ncA_LIMIT
          controller = ncON
        parameter[2]:
          decel_ramp = ncA_LIMIT
          controller = ncON
        parameter[3]:
          decel_ramp = ncA_LIMIT
          controller = ncON
        quickstop:
          decel_ramp = ncA_LIMIT
        drive_error:
          decel_ramp = ncA_LIMIT
      homing:
        parameter:
          s = 25400
          v_switch = 1000
          v_trigger = 50
          a = 50000
          mode = ncSWITCH_GATE
          edge_sw = ncPOSITIVE
          start_dir = ncPOSITIVE
          trigg_dir = ncPOSITIVE
          ref_pulse = ncOFF
          fix_dir = ncOFF
          tr_s_block = 0
          torque_lim = 0
          ds_block = 0
          ds_stop = 0
      basis:
        parameter:
          v_pos = 10000
          v_neg = 10000
          a1_pos = 50000
          a2_pos = 40000
          a1_neg = 50000
          a2_neg = 40000
    message:
      text:
        parameter:
          format = ncBREAK
          columns = 80
          data_modul = english
```

### Program Logical/Motion/Seam1Array (IEC) - Seamer 1 search control

#### Seam1ArrayCyclic.st - Cyclic code
```iecst
(********************************************************************
 * COPYRIGHT --
 ********************************************************************
 * Program: Seam1Array
 * File: Seam1ArrayCyclic.st
 * Author: Nicke
 * Created: February, 2012
 ********************************************************************
 * Implementation of program Seam1Array
 ********************************************************************)

PROGRAM _INIT

(* Reset search to READY *)
Ax1.Pattern	:= 	READY	;

END_PROGRAM

PROGRAM _CYCLIC
(* cyclic program *)

(* Limit Speed and position of axis*)
	axis1basic.ParaPosition	:= 	LIMIT(Ax1P.AbsMin, axis1basic.ParaPosition, Ax1P.AbsMax)	;
	axis1basic.ParaVelocity	:= 	LIMIT(0, axis1basic.ParaVelocity, 10000)	;

	Ax1.Sensors	:= 	0	; (* Arrange sensor array into a value for determining search pattern *)

IF NOT(Ax1.Active) AND (Control.Achieved1) THEN
	Ax1.Pattern				:= 	READY	;
	Ax1.Count				:= 	0		;
	Ax1.Seek1				:= 	FALSE	;
	Ax1.Seek2				:= 	FALSE	;
	Ax1.SeekFin				:= 	FALSE	;
	Ax1.Text				:=	0		;
	Ax1.StartCheck			:=	FALSE	;
	axis1basic.MoveAbsolute	:= 	FALSE	;
END_IF

IF ((EDGEPOS(Ax1.Seek1) OR EDGEPOS(Ax1.Seek2)) AND (Ax1.Pattern = READY) AND NOT(Ax1.Block)) THEN
	Ax1.Seek2	:= 	FALSE	;
	IF (S81Photo.In) THEN
		Ax1.Sensors	:= 	Ax1.Sensors + 1	;
	END_IF
	IF (S82Photo.In) THEN
 		Ax1.Sensors	:= 	Ax1.Sensors + 2	;
	END_IF
	IF (S83Photo.In) THEN
 		Ax1.Sensors	:= 	Ax1.Sensors + 4	;
	END_IF
	IF (S84Photo.In) THEN
 		Ax1.Sensors	:= 	Ax1.Sensors + 8	;
	END_IF

	IF(axis1basic.ActPosition <= Ax1P.FRAbsMin) AND(Ax1.Sensors = 0) THEN
		Ax1.Sensors	:= 	1	;
	END_IF

	CASE Ax1.Sensors OF (* Determine type of search pattern from sensors *)
	0,8:
		Ax1.Pattern				:= 	FAST_REV		;
		Ax1.Text				:= 	1				;
		axis1basic.ParaPosition	:= 	Ax1P.FRAbsMin	;
		axis1basic.ParaVelocity	:= 	Ax1P.FastSpeed	;
		axis1basic.MoveAbsolute	:= 	TRUE			;
	1,9:
		Ax1.Pattern				:= 	SLOW_REV								;
		Ax1.Text				:= 	2										;
		axis1basic.ParaPosition	:= 	axis1basic.ActPosition - Ax1P.SlowDist	;
		axis1basic.ParaVelocity	:= 	Ax1P.SlowSpeed							;
		IF (axis1basic.ParaPosition < Ax1P.AbsMin) THEN (* If calculated position is outside operating area, substitute minimum position for calculated value *)
			axis1basic.ParaPosition	:= 	Ax1P.AbsMin	;
		END_IF
		axis1basic.MoveAbsolute	:= 	TRUE		;
	2,3,10,11:
		Ax1.Pattern				:= 	CHECK									;
		Ax1.Text				:= 	3										;
		Ax1.StartCheck			:=	TRUE	;
		axis1basic.ParaPosition	:= 	axis1basic.ActPosition + Ax1P.FCDist	; (* Forward direction for search *)
		axis1basic.ParaVelocity	:= 	Ax1P.FCSpeed							;
		IF (axis1basic.ParaPosition > (Ax1P.AbsMax + 200)) THEN (* If calculated position is outside operating area, substitute maximum position for calculated value *)
				axis1basic.ParaPosition	:= 	(Ax1P.AbsMax + 200)	;
		END_IF
		axis1basic.MoveAbsolute	:= 	TRUE		;
	4..7:
		Ax1.Pattern				:= 	SLOW_FWD								;
		Ax1.Text				:= 	4										;
		axis1basic.ParaPosition	:= 	axis1basic.ActPosition + Ax1P.SlowDist	;
		axis1basic.ParaVelocity	:= 	Ax1P.SlowSpeed							;
		IF axis1basic.ParaPosition > Ax1P.AbsMax THEN (* If calculated position is outside operating area, substitute maximum position for calculated value *)
			axis1basic.ParaPosition	:= 	Ax1P.AbsMax	;
		END_IF
		axis1basic.MoveAbsolute	:= 	TRUE		;
	12..15:
		Ax1.Pattern				:= 	FAST_FWD		;
		Ax1.Text				:= 	5				;
		axis1basic.ParaPosition	:= 	Ax1P.FFAbsMax	;
		axis1basic.ParaVelocity	:= 	Ax1P.FastSpeed	;
		axis1basic.MoveAbsolute	:= 	TRUE			;

	END_CASE

END_IF

(* Cancel movement at EMO *)
IF EDGEPOS(Control.EStop1) AND NOT(axis1basic.StatusDisabled) THEN
	Ax1.Pattern		:= 	0		;
	Ax1.Count		:= 	0		;
//	axis1basic.Stop	:= 	TRUE	;
	axis1basic.MoveAbsolute	:=	FALSE	;
END_IF

CASE Ax1.Pattern OF
FAST_REV: (**** FAST_ REV Search Pattern ****)
	IF EDGEPOS(S81Photo.In) THEN (* Check for Rev sensor rising edge *)
		axis1basic.ParaPosition	:= 	axis1basic.ActPosition - Ax1P.RevFeed	;
		IF(axis1basic.ParaPosition < Ax1P.AbsMin) THEN
			axis1basic.ParaPosition	:=	Ax1P.AbsMin	;
		END_IF
		axis1basic.MoveAbsolute	:= 	TRUE									;
	END_IF

SLOW_REV: (**** SLOW_REV Search Pattern ****)
	IF EDGEPOS(S82Photo.In) THEN (* Check for Edge sensor rising edge *)
		axis1basic.ParaPosition	:= 	axis1basic.ActPosition + Ax1P.SlowAdj1	;
		IF(axis1basic.ParaPosition < Ax1P.AbsMin) THEN
			axis1basic.ParaPosition	:=	Ax1P.AbsMin	;
		END_IF
		axis1basic.MoveAbsolute	:= 	TRUE									;
		axis1basic.ParaVelocity	:= 	Ax1P.FCSpeed							;
	END_IF

CHECK: (**** CHECK Search Pattern ****)
	IF EDGENEG(S82Photo.In) THEN (* Check for Edge sensor rising edge *)
		Ax1.CheckPosition		:= 	axis1basic.ActPosition					;
		Ax1.StartCheck			:=	FALSE	;
		axis1basic.ParaPosition	:= 	axis1basic.ActPosition - Ax1P.SlowAdj3	;
		IF(axis1basic.ParaPosition > Ax1P.AbsMax) THEN
			axis1basic.ParaPosition	:=	Ax1P.AbsMax	;
		END_IF
		axis1basic.MoveAbsolute	:= 	TRUE									;
	END_IF
	IF EDGENEG(axis1basic.StatusMotionDiscrete) AND NOT(Ax1.StartCheck) THEN
		Ax1.Count	:= 	Ax1.Count + 1	;
	END_IF

SLOW_FWD: (**** SLOW_FWD Search Pattern ****)
	IF EDGENEG(S83Photo.In) THEN (* Check for Edge sensor rising edge *)
		axis1basic.ParaPosition	:= 	axis1basic.ActPosition - Ax1P.SlowAdj2	;
		IF(axis1basic.ParaPosition > Ax1P.AbsMax) THEN
			axis1basic.ParaPosition	:=	Ax1P.AbsMax	;
		END_IF
		axis1basic.ParaVelocity	:= 	Ax1P.FCSpeed							;
		axis1basic.MoveAbsolute	:= 	TRUE									;
	END_IF

FAST_FWD: (**** FAST_FWD Search Pattern ****)
	IF EDGENEG(S84Photo.In) THEN (* Check for Fwd sensor falling edge *)
		axis1basic.ParaPosition	:= 	axis1basic.ActPosition + Ax1P.FwdFeed	;
		IF(axis1basic.ParaPosition > Ax1P.AbsMax) THEN
			axis1basic.ParaPosition	:=	Ax1P.AbsMax	;
		END_IF
		axis1basic.MoveAbsolute	:= 	TRUE									;
	END_IF

END_CASE

IF EDGENEG(axis1basic.StatusMotionDiscrete) AND (Ax1.Pattern > READY) THEN (* Reset Search Pattern *)
	Ax1.Pattern		:= 	READY	;
	Ax1.Text		:= 	0		;
	Ax1.Seek2		:= 	TRUE	;
	Ax1.StartCheck	:=	FALSE	;
	CASE Ax1.Count OF
		2: 	Ax1.Count	:= 	0						;
			Ax1.SeekFin	:= 	TRUE					;
			Ax1.Seek2	:= 	FALSE					;
			Ax1.Measure	:= 	axis1basic.ActPosition	;
	END_CASE
END_IF

(*Enable screen reset button during drive error*)
IF (Ax1.Error) THEN
	Ax1.ResetEnable	:= 	SHOW	;
ELSE
	Ax1.ResetEnable	:= 	HIDE	;
END_IF

(* If actual position is outside operating area then stop output *)
IF ((axis1basic.ActPosition > (Ax1P.AbsMax + 100)) OR (axis1basic.ActPosition < (Ax1P.AbsMin - 200))) AND (Ax1.OriginSet) AND NOT(axis1basic.StatusDisabled) THEN
	axis1basic.Stop	:= 	TRUE	;
END_IF

(* Copy actual positon for flip up arm calculations *)
ArmsTemp1.ActPos	:=	axis1basic.ActPosition	;

END_PROGRAM
```

### Program Logical/Motion/Axis1State (IEC)

#### Axis1StateInit.ld
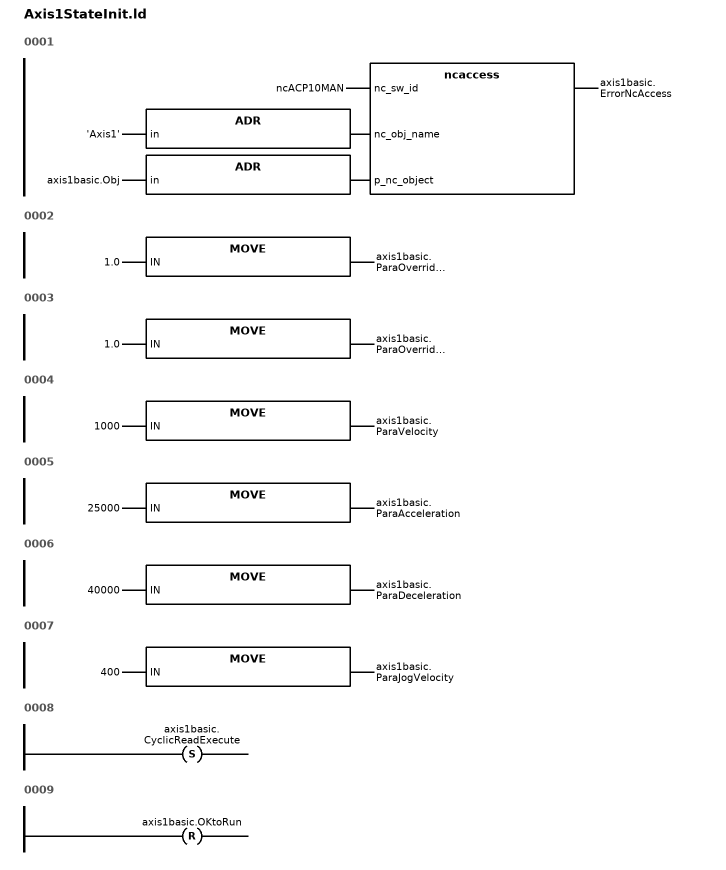
Ladder, written as Structured Text:
```iecst
PROGRAM _INIT
(* Network 1 *)
axis1basic.ErrorNcAccess := ncaccess(nc_sw_id := ncACP10MAN, nc_obj_name := ADR(in := 'Axis1'), p_nc_object := ADR(in := axis1basic.Obj));

(* Network 2 *)
axis1basic.ParaOverrideVelocity := 1.0;

(* Network 3 *)
axis1basic.ParaOverrideAcceleration := 1.0;

(* Network 4 *)
axis1basic.ParaVelocity := 1000;

(* Network 5 *)
axis1basic.ParaAcceleration := 25000;

(* Network 6 *)
axis1basic.ParaDeceleration := 40000;

(* Network 7 *)
axis1basic.ParaJogVelocity := 400;

(* Network 8 *)
axis1basic.CyclicReadExecute := TRUE;

(* Network 9 *)
axis1basic.OKtoRun := FALSE;
END_PROGRAM
```

#### Axis1StateCyclic.ld
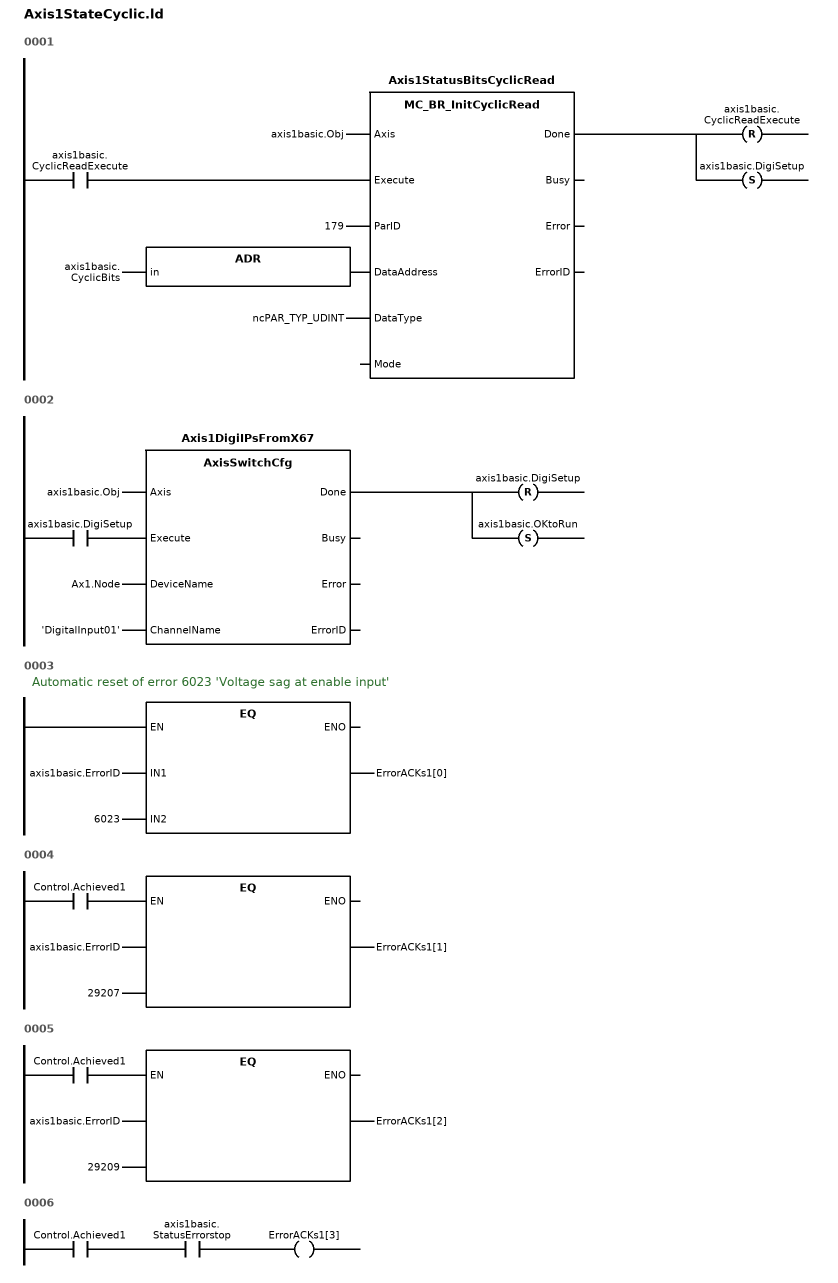
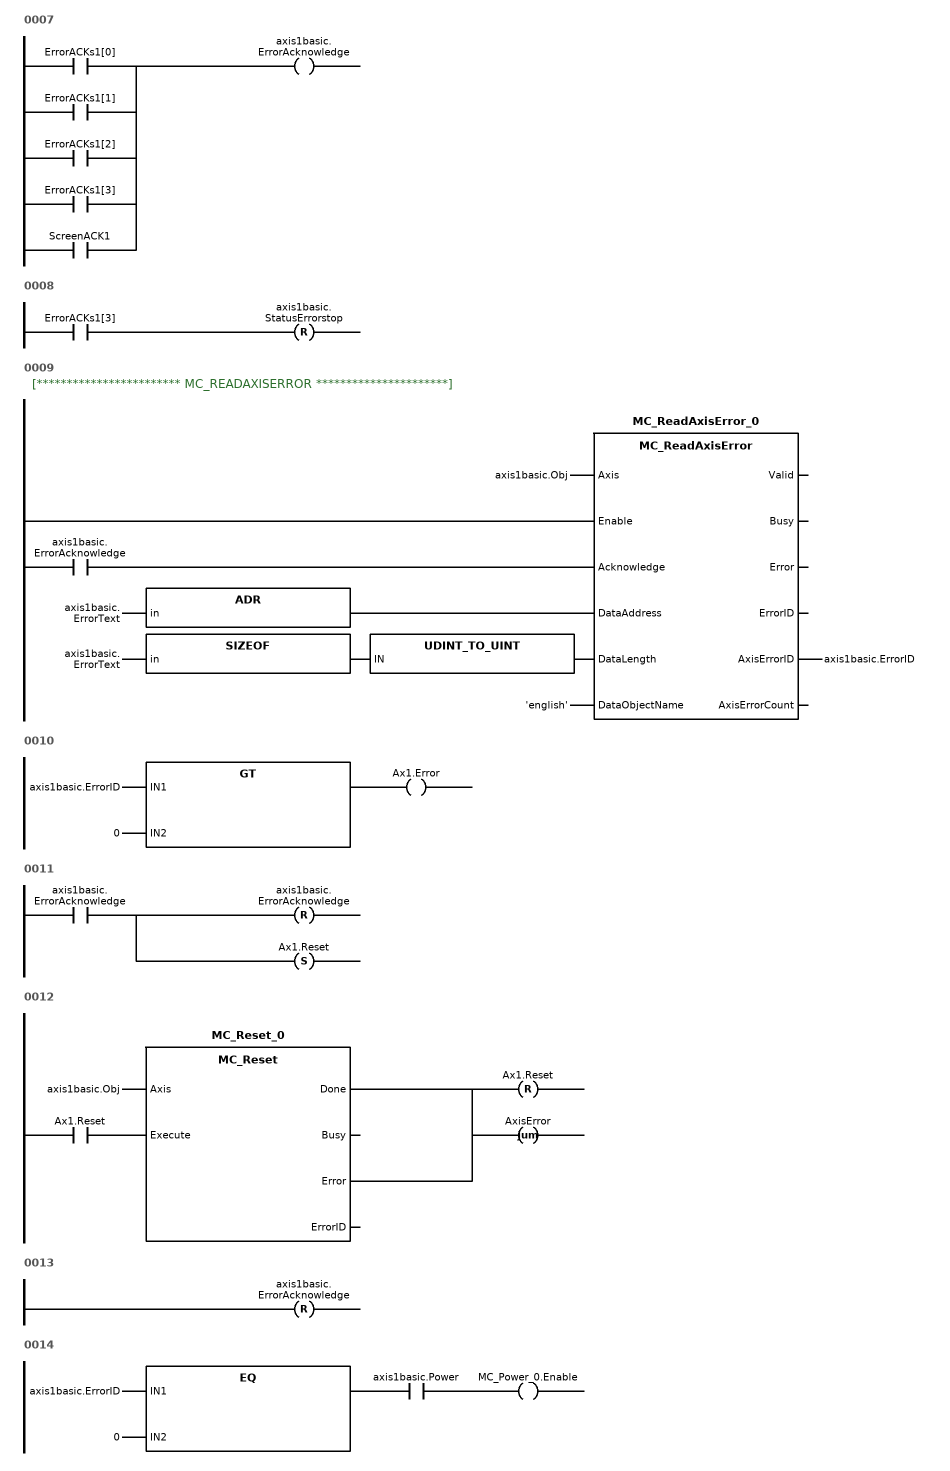
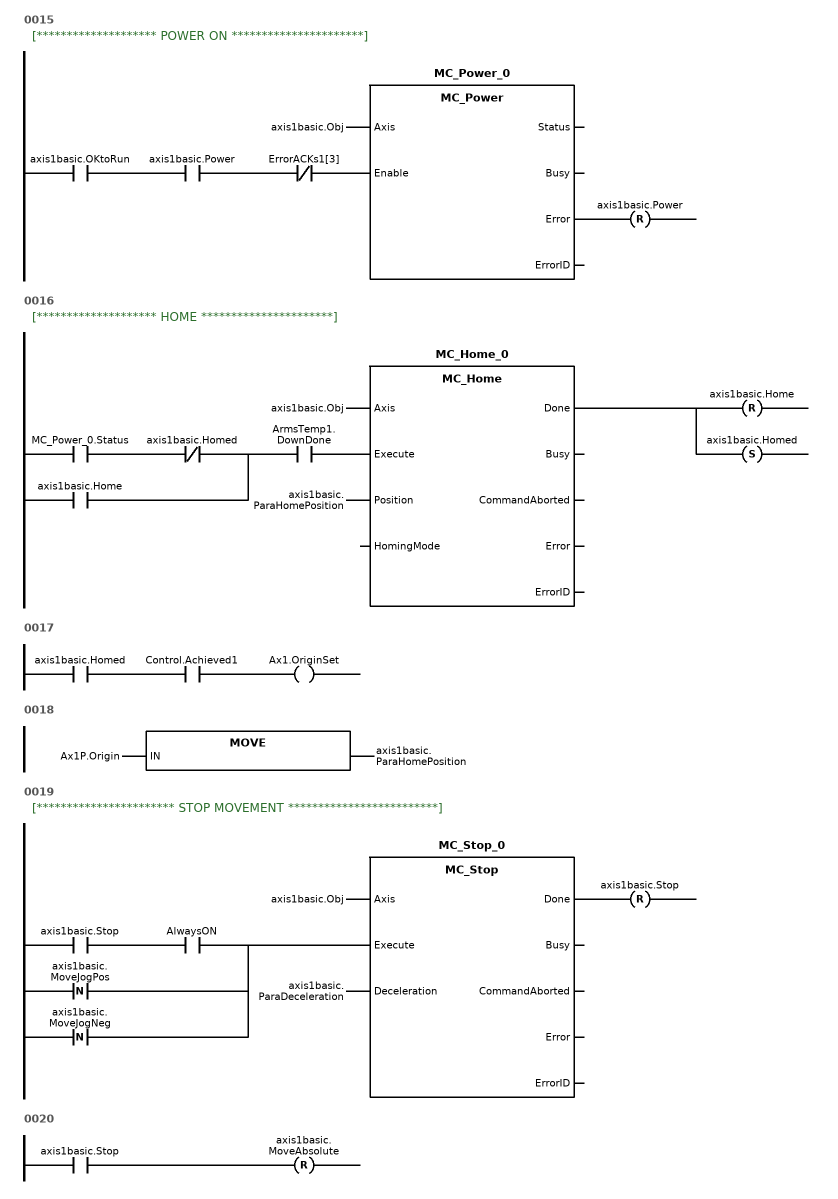
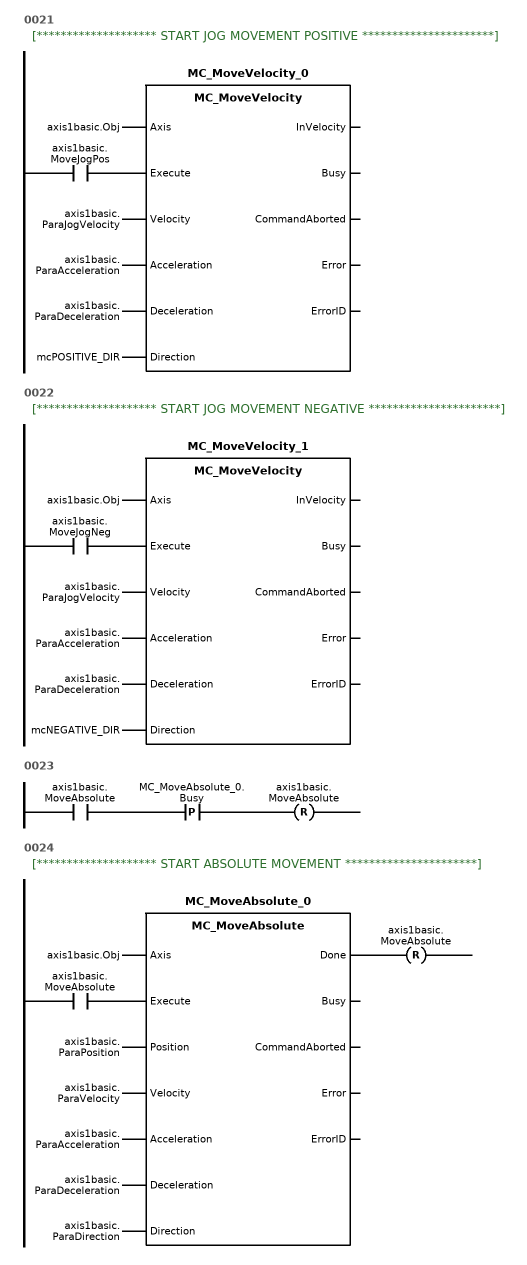
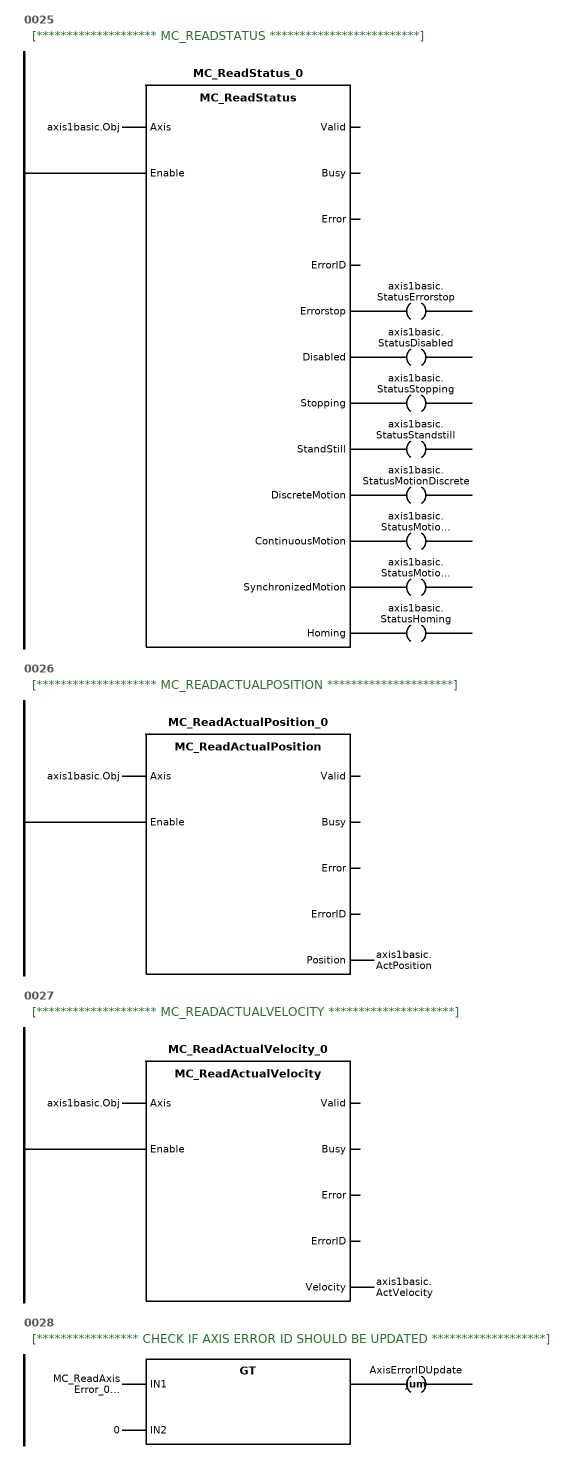
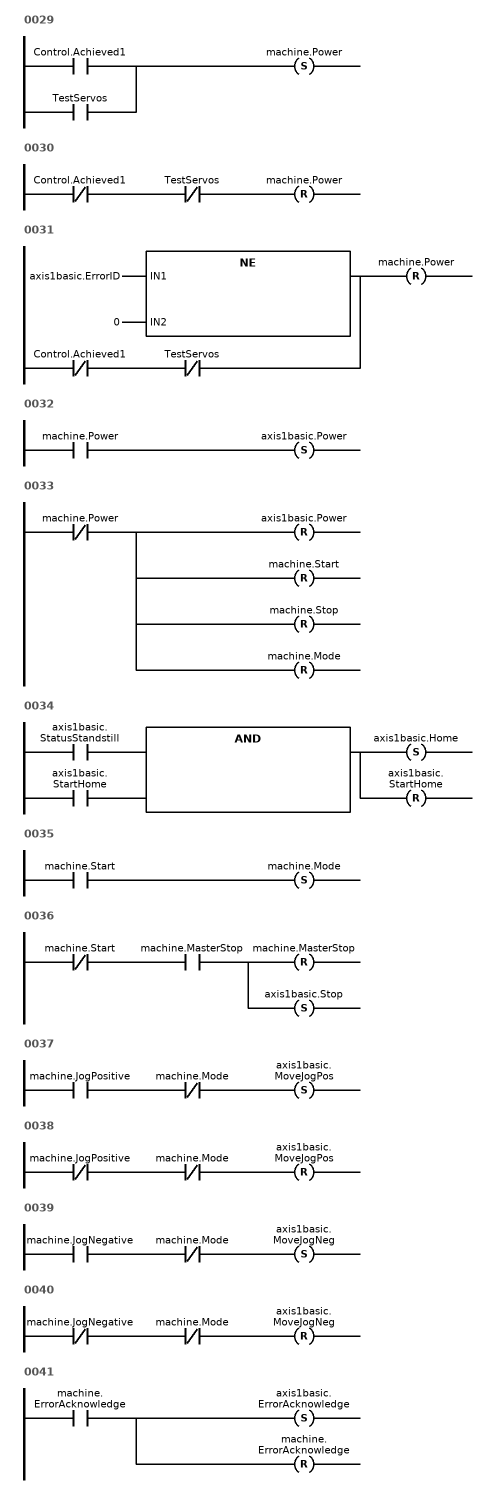
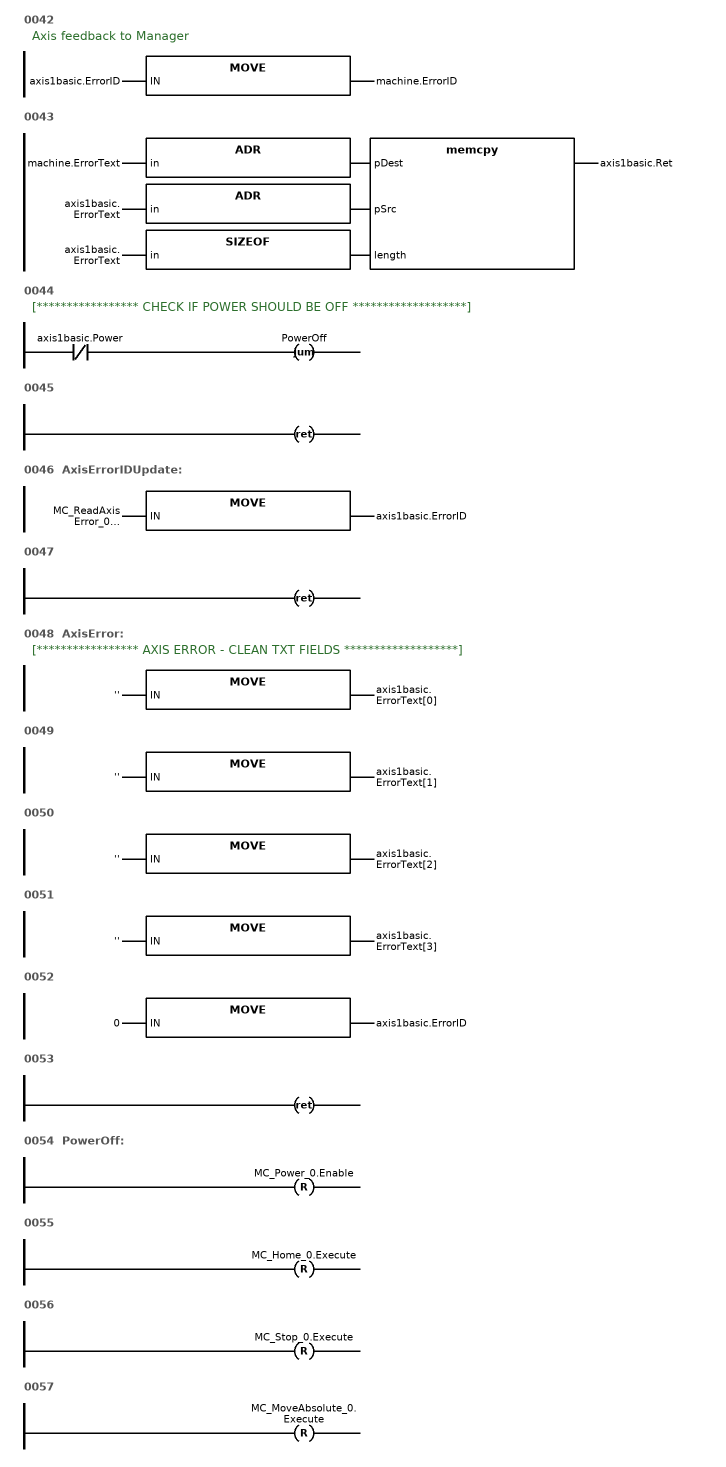
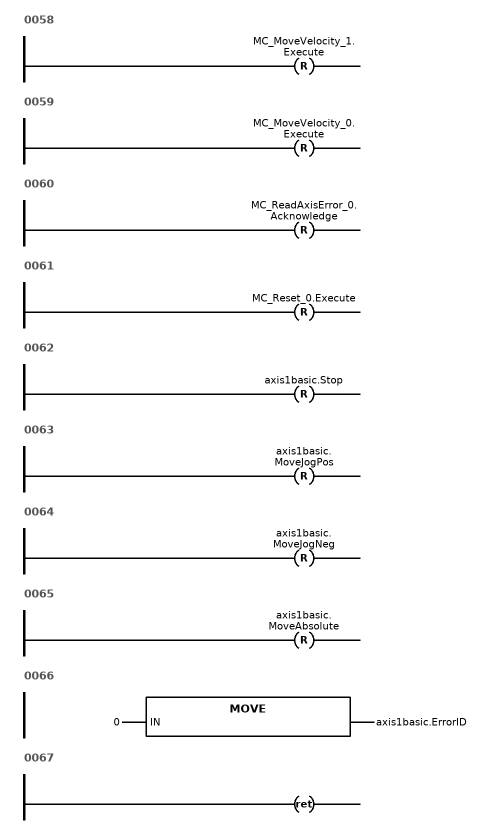
Ladder, written as Structured Text:
```iecst
PROGRAM _CYCLIC
VAR
    _p1 : BOOL;
    _e2 : F_TRIG;
    _e3 : F_TRIG;
    _e4 : R_TRIG;
    _p5 : BOOL;
    _t6 : BOOL;
    _p7 : BOOL;
END_VAR
(* Network 1 *)
Axis1StatusBitsCyclicRead(Axis := axis1basic.Obj, Execute := axis1basic.CyclicReadExecute, ParID := 179, DataAddress := ADR(in := axis1basic.CyclicBits), DataType := ncPAR_TYP_UDINT);
IF Axis1StatusBitsCyclicRead.Done THEN
    axis1basic.CyclicReadExecute := FALSE;
    axis1basic.DigiSetup := TRUE;
END_IF;

(* Network 2 *)
Axis1DigiIPsFromX67(Axis := axis1basic.Obj, Execute := axis1basic.DigiSetup, DeviceName := Ax1.Node, ChannelName := 'DigitalInput01');
IF Axis1DigiIPsFromX67.Done THEN
    axis1basic.DigiSetup := FALSE;
    axis1basic.OKtoRun := TRUE;
END_IF;

(* Network 3: Automatic reset of error 6023 'Voltage sag at enable input' *)
ErrorACKs1[0] := axis1basic.ErrorID = 6023;

(* Network 4 *)
IF Control.Achieved1 THEN ErrorACKs1[1] := axis1basic.ErrorID = 29207; END_IF;

(* Network 5 *)
IF Control.Achieved1 THEN ErrorACKs1[2] := axis1basic.ErrorID = 29209; END_IF;

(* Network 6 *)
ErrorACKs1[3] := Control.Achieved1 AND axis1basic.StatusErrorstop;

(* Network 7 *)
axis1basic.ErrorAcknowledge := ErrorACKs1[0] OR ErrorACKs1[1] OR ErrorACKs1[2] OR ErrorACKs1[3] OR ScreenACK1;

(* Network 8 *)
IF ErrorACKs1[3] THEN axis1basic.StatusErrorstop := FALSE; END_IF;

(* Network 9: [************************ MC_READAXISERROR **********************] *)
MC_ReadAxisError_0(Axis := axis1basic.Obj, Enable := TRUE, Acknowledge := axis1basic.ErrorAcknowledge, DataAddress := ADR(in := axis1basic.ErrorText), DataLength := UDINT_TO_UINT(SIZEOF(in := axis1basic.ErrorText)), DataObjectName := 'english');
axis1basic.ErrorID := MC_ReadAxisError_0.AxisErrorID;

(* Network 10 *)
Ax1.Error := axis1basic.ErrorID > 0;

(* Network 11 *)
_p1 := axis1basic.ErrorAcknowledge;
IF axis1basic.ErrorAcknowledge THEN axis1basic.ErrorAcknowledge := FALSE; END_IF;
IF _p1 THEN Ax1.Reset := TRUE; END_IF;

(* Network 12 *)
MC_Reset_0(Axis := axis1basic.Obj, Execute := Ax1.Reset);
IF MC_Reset_0.Done OR MC_Reset_0.Error THEN
    Ax1.Reset := FALSE;
    JMP AxisError;
END_IF;

(* Network 13 *)
axis1basic.ErrorAcknowledge := FALSE;

(* Network 14 *)
MC_Power_0.Enable := (axis1basic.ErrorID = 0) AND axis1basic.Power;

(* Network 15: [******************** POWER ON **********************] *)
MC_Power_0(Axis := axis1basic.Obj, Enable := axis1basic.OKtoRun AND axis1basic.Power AND NOT ErrorACKs1[3]);
IF MC_Power_0.Error THEN axis1basic.Power := FALSE; END_IF;

(* Network 16: [******************** HOME **********************] *)
MC_Home_0(Axis := axis1basic.Obj, Execute := ((MC_Power_0.Status AND NOT axis1basic.Homed) OR axis1basic.Home) AND ArmsTemp1.DownDone, Position := axis1basic.ParaHomePosition);
IF MC_Home_0.Done THEN
    axis1basic.Home := FALSE;
    axis1basic.Homed := TRUE;
END_IF;

(* Network 17 *)
Ax1.OriginSet := axis1basic.Homed AND Control.Achieved1;

(* Network 18 *)
axis1basic.ParaHomePosition := Ax1P.Origin;

(* Network 19: [*********************** STOP MOVEMENT *************************] *)
_e2(CLK := axis1basic.MoveJogPos);
_e3(CLK := axis1basic.MoveJogNeg);
MC_Stop_0(Axis := axis1basic.Obj, Execute := (axis1basic.Stop AND AlwaysON) OR _e2.Q OR _e3.Q, Deceleration := axis1basic.ParaDeceleration);
IF MC_Stop_0.Done THEN axis1basic.Stop := FALSE; END_IF;

(* Network 20 *)
IF axis1basic.Stop THEN axis1basic.MoveAbsolute := FALSE; END_IF;

(* Network 21: [******************** START JOG MOVEMENT POSITIVE **********************] *)
MC_MoveVelocity_0(Axis := axis1basic.Obj, Execute := axis1basic.MoveJogPos, Velocity := axis1basic.ParaJogVelocity, Acceleration := axis1basic.ParaAcceleration, Deceleration := axis1basic.ParaDeceleration, Direction := mcPOSITIVE_DIR);

(* Network 22: [******************** START JOG MOVEMENT NEGATIVE **********************] *)
MC_MoveVelocity_1(Axis := axis1basic.Obj, Execute := axis1basic.MoveJogNeg, Velocity := axis1basic.ParaJogVelocity, Acceleration := axis1basic.ParaAcceleration, Deceleration := axis1basic.ParaDeceleration, Direction := mcNEGATIVE_DIR);

(* Network 23 *)
_e4(CLK := MC_MoveAbsolute_0.Busy);
IF axis1basic.MoveAbsolute AND _e4.Q THEN axis1basic.MoveAbsolute := FALSE; END_IF;

(* Network 24: [******************** START ABSOLUTE MOVEMENT **********************] *)
MC_MoveAbsolute_0(Axis := axis1basic.Obj, Execute := axis1basic.MoveAbsolute, Position := axis1basic.ParaPosition, Velocity := axis1basic.ParaVelocity, Acceleration := axis1basic.ParaAcceleration, Deceleration := axis1basic.ParaDeceleration, Direction := axis1basic.ParaDirection);
IF MC_MoveAbsolute_0.Done THEN axis1basic.MoveAbsolute := FALSE; END_IF;

(* Network 25: [******************** MC_READSTATUS *************************] *)
MC_ReadStatus_0(Axis := axis1basic.Obj, Enable := TRUE);
axis1basic.StatusErrorstop := MC_ReadStatus_0.Errorstop;
axis1basic.StatusDisabled := MC_ReadStatus_0.Disabled;
axis1basic.StatusStopping := MC_ReadStatus_0.Stopping;
axis1basic.StatusStandstill := MC_ReadStatus_0.StandStill;
axis1basic.StatusMotionDiscrete := MC_ReadStatus_0.DiscreteMotion;
axis1basic.StatusMotionContinous := MC_ReadStatus_0.ContinuousMotion;
axis1basic.StatusMotionSynchronized := MC_ReadStatus_0.SynchronizedMotion;
axis1basic.StatusHoming := MC_ReadStatus_0.Homing;

(* Network 26: [******************** MC_READACTUALPOSITION *********************] *)
MC_ReadActualPosition_0(Axis := axis1basic.Obj, Enable := TRUE);
axis1basic.ActPosition := MC_ReadActualPosition_0.Position;

(* Network 27: [******************** MC_READACTUALVELOCITY *********************] *)
MC_ReadActualVelocity_0(Axis := axis1basic.Obj, Enable := TRUE);
axis1basic.ActVelocity := MC_ReadActualVelocity_0.Velocity;

(* Network 28: [***************** CHECK IF AXIS ERROR ID SHOULD BE UPDATED *******************] *)
IF MC_ReadAxisError_0.AxisErrorID > 0 THEN JMP AxisErrorIDUpdate; END_IF;

(* Network 29 *)
IF Control.Achieved1 OR TestServos THEN machine.Power := TRUE; END_IF;

(* Network 30 *)
IF NOT Control.Achieved1 AND NOT TestServos THEN machine.Power := FALSE; END_IF;

(* Network 31 *)
IF (NOT Control.Achieved1 AND NOT TestServos) OR (axis1basic.ErrorID <> 0) THEN
    machine.Power := FALSE;
END_IF;

(* Network 32 *)
IF machine.Power THEN axis1basic.Power := TRUE; END_IF;

(* Network 33 *)
IF NOT machine.Power THEN axis1basic.Power := FALSE; END_IF;
_p5 := NOT machine.Power;
IF NOT machine.Power THEN machine.Start := FALSE; END_IF;
IF _p5 THEN
    machine.Stop := FALSE;
    machine.Mode := FALSE;
END_IF;

(* Network 34 *)
_t6 := axis1basic.StatusStandstill AND axis1basic.StartHome;
IF _t6 THEN
    axis1basic.Home := TRUE;
    axis1basic.StartHome := FALSE;
END_IF;

(* Network 35 *)
IF machine.Start THEN machine.Mode := TRUE; END_IF;

(* Network 36 *)
_p7 := NOT machine.Start AND machine.MasterStop;
IF NOT machine.Start AND machine.MasterStop THEN machine.MasterStop := FALSE; END_IF;
IF _p7 THEN axis1basic.Stop := TRUE; END_IF;

(* Network 37 *)
IF machine.JogPositive AND NOT machine.Mode THEN axis1basic.MoveJogPos := TRUE; END_IF;

(* Network 38 *)
IF NOT machine.JogPositive AND NOT machine.Mode THEN axis1basic.MoveJogPos := FALSE; END_IF;

(* Network 39 *)
IF machine.JogNegative AND NOT machine.Mode THEN axis1basic.MoveJogNeg := TRUE; END_IF;

(* Network 40 *)
IF NOT machine.JogNegative AND NOT machine.Mode THEN axis1basic.MoveJogNeg := FALSE; END_IF;

(* Network 41 *)
IF machine.ErrorAcknowledge THEN
    axis1basic.ErrorAcknowledge := TRUE;
    machine.ErrorAcknowledge := FALSE;
END_IF;

(* Network 42: Axis feedback to Manager *)
machine.ErrorID := axis1basic.ErrorID;

(* Network 43 *)
axis1basic.Ret := memcpy(pDest := ADR(in := machine.ErrorText), pSrc := ADR(in := axis1basic.ErrorText), length := SIZEOF(in := axis1basic.ErrorText));

(* Network 44: [***************** CHECK IF POWER SHOULD BE OFF *******************] *)
IF NOT axis1basic.Power THEN JMP PowerOff; END_IF;

(* Network 45 *)
RETURN;

(* Network 46 *)
AxisErrorIDUpdate:
axis1basic.ErrorID := MC_ReadAxisError_0.AxisErrorID;

(* Network 47 *)
RETURN;

(* Network 48: [***************** AXIS ERROR - CLEAN TXT FIELDS *******************] *)
AxisError:
axis1basic.ErrorText[0] := '';

(* Network 49 *)
axis1basic.ErrorText[1] := '';

(* Network 50 *)
axis1basic.ErrorText[2] := '';

(* Network 51 *)
axis1basic.ErrorText[3] := '';

(* Network 52 *)
axis1basic.ErrorID := 0;

(* Network 53 *)
RETURN;

(* Network 54 *)
PowerOff:
MC_Power_0.Enable := FALSE;

(* Network 55 *)
MC_Home_0.Execute := FALSE;

(* Network 56 *)
MC_Stop_0.Execute := FALSE;

(* Network 57 *)
MC_MoveAbsolute_0.Execute := FALSE;

(* Network 58 *)
MC_MoveVelocity_1.Execute := FALSE;

(* Network 59 *)
MC_MoveVelocity_0.Execute := FALSE;

(* Network 60 *)
MC_ReadAxisError_0.Acknowledge := FALSE;

(* Network 61 *)
MC_Reset_0.Execute := FALSE;

(* Network 62 *)
axis1basic.Stop := FALSE;

(* Network 63 *)
axis1basic.MoveJogPos := FALSE;

(* Network 64 *)
axis1basic.MoveJogNeg := FALSE;

(* Network 65 *)
axis1basic.MoveAbsolute := FALSE;

(* Network 66 *)
axis1basic.ErrorID := 0;

(* Network 67 *)
RETURN;
END_PROGRAM
```

### Program Logical/Motion/Seam2Array (IEC) - A new program

#### Seam2ArrayCyclic.st - Cyclic code
```iecst
(********************************************************************
 * COPYRIGHT --
 ********************************************************************
 * Program: Seam2Array
 * File: Seam2ArrayCyclic.st
 * Author: NickE
 * Created: February, 2012
 ********************************************************************
 * Implementation of program Seam2Array
 ********************************************************************)

PROGRAM _INIT

(* Reset search to READY *)
Ax2.Pattern	:= 	READY	;

END_PROGRAM

PROGRAM _CYCLIC
(* cyclic program *)

(* Limit Speed and position of axis*)
	axis2basic.ParaPosition	:= 	LIMIT(Ax2P.AbsMin, axis2basic.ParaPosition, Ax2P.AbsMax)	;
	axis2basic.ParaVelocity	:= 	LIMIT(0, axis2basic.ParaVelocity, 10000)	;

	Ax2.Sensors	:= 	0	; (* Arrange sensor array into a value for determining search pattern *)

	IF NOT(Ax2.Active) AND (Control.Achieved1) THEN
	Ax2.Pattern				:= 	READY	;
	Ax2.Count				:= 	0		;
	Ax2.Seek1				:= 	FALSE	;
	Ax2.Seek2				:= 	FALSE	;
	Ax2.SeekFin				:= 	FALSE	;
	Ax2.Text				:=	0		;
	Ax2.StartCheck			:=	FALSE	;
	axis2basic.MoveAbsolute	:= 	FALSE	;
END_IF

IF ((EDGEPOS(Ax2.Seek1) OR EDGEPOS(Ax2.Seek2)) AND (Ax2.Pattern = READY) AND NOT(Ax2.Block)) THEN
	Ax2.Seek2	:= 	FALSE	;
	IF (S91Photo.In) THEN
		Ax2.Sensors	:= 	Ax2.Sensors + 1	;
	END_IF
	IF (S92Photo.In) THEN
 		Ax2.Sensors	:= 	Ax2.Sensors + 2	;
	END_IF
	IF (S93Photo.In) THEN
 		Ax2.Sensors	:= 	Ax2.Sensors + 4	;
	END_IF
	IF (S94Photo.In) THEN
 		Ax2.Sensors	:= 	Ax2.Sensors + 8	;
	END_IF

	IF(axis2basic.ActPosition <= Ax2P.FRAbsMin) AND(Ax2.Sensors = 0) THEN
		Ax2.Sensors	:= 	1	;
	END_IF

	CASE Ax2.Sensors OF (* Determine type of search pattern from sensors *)
	0,8:
		Ax2.Pattern				:= 	FAST_REV		;
		Ax2.Text				:= 	1				;
		axis2basic.ParaPosition	:= 	Ax2P.FRAbsMin	;
		axis2basic.ParaVelocity	:= 	Ax2P.FastSpeed	;
		axis2basic.MoveAbsolute	:= 	TRUE			;
	1,9:
		Ax2.Pattern				:= 	SLOW_REV								;
		Ax2.Text				:= 	2										;
		axis2basic.ParaPosition	:= 	axis2basic.ActPosition - Ax2P.SlowDist	;
		axis2basic.ParaVelocity	:= 	Ax2P.SlowSpeed							;
		IF (axis2basic.ParaPosition < Ax2P.AbsMin) THEN (* If calculated position is outside operating area, substitute minimum position for calculated value *)
			axis2basic.ParaPosition	:= 	Ax2P.AbsMin	;
		END_IF
		axis2basic.MoveAbsolute	:= 	TRUE	;
	2,3,10,11:
		Ax2.Pattern				:= 	CHECK									;
		Ax2.Text				:= 	3										;
		Ax2.StartCheck			:=	TRUE									;
		axis2basic.ParaPosition	:= 	axis2basic.ActPosition + Ax2P.FCDist	; (* Forward direction for search *)
		axis2basic.ParaVelocity	:= 	Ax2P.FCSpeed							;
		IF (axis2basic.ParaPosition > (Ax2P.AbsMax + 200)) THEN (* If calculated position is outside operating area, substitute maximum position for calculated value *)
				axis2basic.ParaPosition	:= 	(Ax2P.AbsMax + 200)	;
		END_IF
		axis2basic.MoveAbsolute	:= 	TRUE	;
	4..7:
		Ax2.Pattern				:= 	SLOW_FWD								;
		Ax2.Text				:= 	4										;
		axis2basic.ParaPosition	:= 	axis2basic.ActPosition + Ax2P.SlowDist	;
		axis2basic.ParaVelocity	:= 	Ax2P.SlowSpeed							;
		IF axis2basic.ParaPosition > Ax2P.AbsMax THEN (* If calculated position is outside operating area, substitute maximum position for calculated value *)
			axis2basic.ParaPosition	:= 	Ax2P.AbsMax	;
		END_IF
		axis2basic.MoveAbsolute	:= 	TRUE	;
	12..15:
		Ax2.Pattern				:= 	FAST_FWD		;
		Ax2.Text				:= 	5				;
		axis2basic.ParaPosition	:= 	Ax2P.FFAbsMax	;
		axis2basic.ParaVelocity	:= 	Ax2P.FastSpeed	;
		axis2basic.MoveAbsolute	:= 	TRUE			;
	END_CASE

END_IF

(* Cancel movement and capture position at EMO *)
IF EDGEPOS(Control.EStop1) AND NOT(axis2basic.StatusDisabled) THEN
	Ax2.Pattern		:= 	0		;
	Ax2.Count		:= 	0		;
//	axis2basic.Stop	:= 	TRUE	;
	axis2basic.MoveAbsolute	:=	FALSE	;
END_IF

CASE Ax2.Pattern OF
FAST_REV: (**** FAST_ REV Search Pattern ****)
	IF EDGEPOS(S91Photo.In) THEN (* Check for Rev sensor rising edge *)
		axis2basic.ParaPosition	:= 	axis2basic.ActPosition - Ax2P.RevFeed	;
		IF(axis2basic.ParaPosition < Ax2P.AbsMin) THEN
			axis2basic.ParaPosition	:=	Ax2P.AbsMin	;
		END_IF
		axis2basic.MoveAbsolute	:= 	TRUE									;
	END_IF

SLOW_REV: (**** SLOW_REV Search Pattern ****)
	IF EDGEPOS(S92Photo.In) THEN (* Check for Edge sensor rising edge *)
		axis2basic.ParaPosition	:= 	axis2basic.ActPosition + Ax2P.SlowAdj1	;
		IF(axis2basic.ParaPosition < Ax2P.AbsMin) THEN
			axis2basic.ParaPosition	:=	Ax2P.AbsMin	;
		END_IF
		axis2basic.MoveAbsolute	:= 	TRUE									;
		axis2basic.ParaVelocity	:= 	Ax2P.FCSpeed							;
	END_IF

CHECK: (**** CHECK Search Pattern ****)
	IF EDGENEG(S92Photo.In) THEN (* Check for Edge sensor rising edge *)
		Ax2.CheckPosition		:= 	axis2basic.ActPosition					;
		axis2basic.ParaPosition	:= 	axis2basic.ActPosition - Ax2P.SlowAdj3	;
		Ax2.StartCheck			:=	FALSE	;
		IF(axis2basic.ParaPosition > Ax2P.AbsMax) THEN
			axis2basic.ParaPosition	:=	Ax2P.AbsMax	;
		END_IF
		axis2basic.MoveAbsolute	:= 	TRUE									;
	END_IF
	IF EDGENEG(axis2basic.StatusMotionDiscrete) AND NOT(Ax2.StartCheck) THEN
		Ax2.Count	:= 	Ax2.Count + 1	;
	END_IF

SLOW_FWD: (**** SLOW_FWD Search Pattern ****)
	IF EDGENEG(S93Photo.In) THEN (* Check for Edge sensor rising edge *)
		axis2basic.ParaPosition	:= 	axis2basic.ActPosition - Ax2P.SlowAdj2	;
		IF(axis2basic.ParaPosition > Ax2P.AbsMax) THEN
			axis2basic.ParaPosition	:=	Ax2P.AbsMax	;
		END_IF
		axis2basic.ParaVelocity	:= 	Ax2P.FCSpeed							;
		axis2basic.MoveAbsolute	:= 	TRUE									;
	END_IF

FAST_FWD: (**** FAST_FWD Search Pattern ****)
	IF EDGENEG(S94Photo.In) THEN (* Check for Fwd sensor falling edge *)
		axis2basic.ParaPosition	:= 	axis2basic.ActPosition + Ax2P.FwdFeed	;
		IF(axis2basic.ParaPosition > Ax2P.AbsMax) THEN
			axis2basic.ParaPosition	:=	Ax2P.AbsMax	;
		END_IF
		axis2basic.MoveAbsolute	:= 	TRUE									;
	END_IF

END_CASE

IF EDGENEG(axis2basic.StatusMotionDiscrete) AND (Ax2.Pattern > READY) THEN (* Reset Search Pattern *)
	Ax2.Pattern	:= 	READY	;
	Ax2.Text	:= 	0		;
	Ax2.Seek2	:= 	TRUE	;
	Ax1.StartCheck	:=	FALSE	;
	CASE Ax2.Count OF
		2:	Ax2.Count	:= 	0						;
			Ax2.SeekFin	:= 	TRUE					;
			Ax2.Seek2	:= 	FALSE					;
			Ax2.Measure	:= 	axis2basic.ActPosition	;
	END_CASE
END_IF

(*Enable screen reset button during drive error*)
IF (Ax2.Error) THEN
	Ax2.ResetEnable	:= 	SHOW	;
ELSE
	Ax2.ResetEnable	:= 	HIDE	;
END_IF

	IF (Ax3.Error) THEN
		Ax3.ResetEnable	:= 	SHOW	;
	ELSE
		Ax3.ResetEnable	:= 	HIDE	;
	END_IF

(* If actual position is outside operating area then stop output *)
IF ((axis2basic.ActPosition > (Ax2P.AbsMax + 100)) OR (axis2basic.ActPosition < (Ax2P.AbsMin - 200))) AND (Ax2.OriginSet) AND NOT(axis2basic.StatusDisabled) THEN
	axis2basic.Stop	:= 	TRUE	;
END_IF

(* Copy actual positon for flip up arm calculations *)
ArmsTemp2.ActPos	:=	axis2basic.ActPosition	;

END_PROGRAM
```

### Program Logical/Motion/Axis2State (IEC)

#### Axis2StateInit.ld
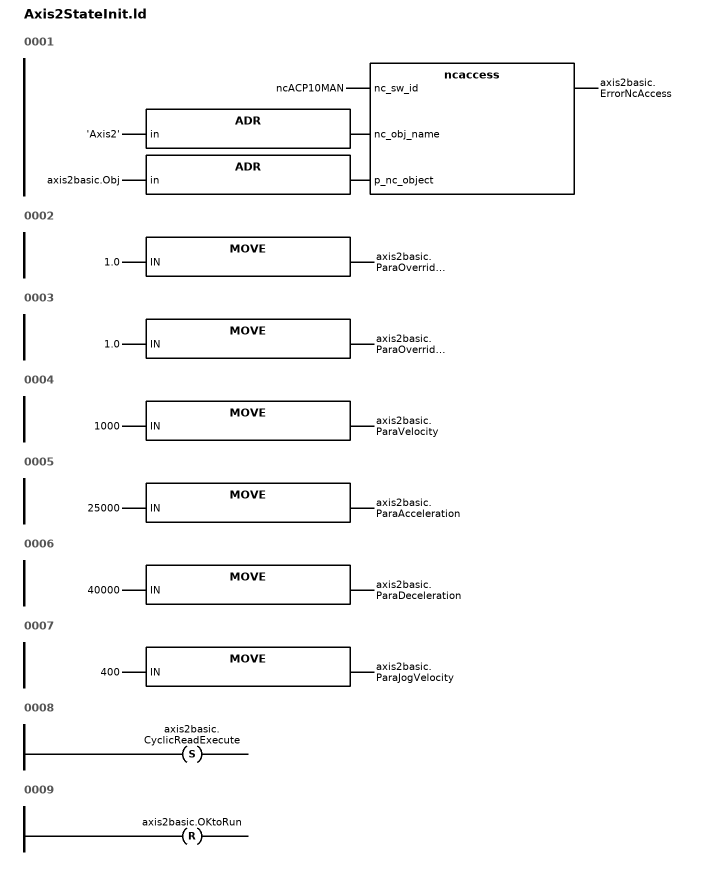
Ladder, written as Structured Text:
```iecst
PROGRAM _INIT
(* Network 1 *)
axis2basic.ErrorNcAccess := ncaccess(nc_sw_id := ncACP10MAN, nc_obj_name := ADR(in := 'Axis2'), p_nc_object := ADR(in := axis2basic.Obj));

(* Network 2 *)
axis2basic.ParaOverrideVelocity := 1.0;

(* Network 3 *)
axis2basic.ParaOverrideAcceleration := 1.0;

(* Network 4 *)
axis2basic.ParaVelocity := 1000;

(* Network 5 *)
axis2basic.ParaAcceleration := 25000;

(* Network 6 *)
axis2basic.ParaDeceleration := 40000;

(* Network 7 *)
axis2basic.ParaJogVelocity := 400;

(* Network 8 *)
axis2basic.CyclicReadExecute := TRUE;

(* Network 9 *)
axis2basic.OKtoRun := FALSE;
END_PROGRAM
```
